	10:// homing sequence
		IF  Stop_PI = 0  THEN
			Out.Homed_PO :=0;
			//check this: reseting expected to match pulse count so that homeing will start if there is a mismatch
			//decide homing direction and homing method //make flag large enough to hit home switch and the limit switch
			IF IN.Limit_NC_NO_CI =0 THEN	//NC switch configuration
				IF bHigh_FI =1 AND bLow_FI =1 THEN	//using normally closed sensor (flag is not on either limit switch)
					IF IN.HomingSet_CI =2 THEN cw := 0; ELSIF IN.HomingSet_CI =3 THEN cw :=1; END_IF //go to high or low first if no limit switch tripped
				END_IF
			ELSE	//NO switch Configuration
				IF bHigh_FI =0 AND bLow_FI =0 THEN	//using normally closed sensor (flag is not on either limit switch)
					IF IN.HomingSet_CI =2 THEN cw := 0; ELSIF IN.HomingSet_CI =3 THEN cw :=1; END_IF //go to high or low first if no limit switch tripped
				END_IF
			END_IF
			//if inputA is hi then turn off (takes 2 cycles to output an increment at cp motor)
				(*if pulses expected = pulse count then do the next move *)
			IF AltSpeedCase = 60 THEN SendPulse(); END_IF
			IF IN.Limit_NC_NO_CI =0 THEN	//NC switch configuration
				IF bHome_FI =0 THEN //use nc switch for sensor [at home position]
					bHomeStart_PI :=0;
					Cancelmove();
					HomeCase := 20;
				END_IF
				ELSE				//NO switch configuration
				IF bHome_FI =1 THEN //use no switch for sensor [at home position]
				bHomeStart_PI :=0;
				Cancelmove();
				HomeCase := 20;
			END_IF	
			END_IF
			(*check this - add in an extra cycle before setting home that moves away from the 
				homed spot in same direction to confirm trigger positino comes on same side of sensor each time*)
		END_IF
	20:	//extra scan before homed
		HomeCase :=50;	//this scan is required to allow for a cancelled move reset after homing
	
	50://after homing reset motor and cancelled bit
		
			Out.Homed_PO := 1;
			//cancelled :=0;	//resets motor after initial homing
			pulsecount :=0;
			expectedPulse :=0;
			Out.DistancePos_PO :=0;
			Out.ExpDistancePos_PO :=0;
			testbool := TRUE;
			HomeCase := 0;	//back to the start
	90://reset to default or?
	
END_CASE
END_METHOD

METHOD PUBLIC InLimits : BOOL
VAR_INPUT
	Req	: REAL;	//reqested degree or position from abs move to be evaluated for limits
END_VAR
//only valid after homing
InLimits := TRUE;
IF IN.SWLimit_Hi_CI <=0 OR IN.SWLimit_Lo_CI >=0 THEN		//check this (may need to have a neg hi at some point)
	//message to say no limits are set
	InLimits :=FALSE;	
END_IF
IF Req <= IN.SWLimit_Hi_CI AND Req >= IN.SWLimit_Lo_CI THEN
	InLimits := TRUE;
	ELSE
		InLimits :=FALSE;
END_IF
END_METHOD

METHOD PUBLIC Jog : BOOL
VAR_INPUT
END_VAR

//add software limits check this
CASE JogCase OF 
	0:	//Main Jog Sequence [Also stops movement]
		IF JogSlow_VI THEN AltspeedReq :=1; ELSE AltSpeedReq :=0;   END_IF
			
		IF JogExecute_VI AND Out.Homed_PO =1  THEN	//if last move is done then allow for manual increment also required to be at home //check sensor check
			IF IN.Limit_NC_NO_CI = 0 THEN	//NC limit switch configuration
				IF bHigh_FI AND bLow_FI THEN //set direction via hmi unless on a limit switch then default to locateposition()
					IF CW_VI = 1 	THEN	CW := 1; 	ELSE CW:=0; 	END_IF
					IF bhigh_fI = 0	THEN 	CW:=0; 		END_IF
					IF bLow_FI = 0 	THEN 	CW:=1; 		END_IF
				END_IF
				ELSE	//NO limit switch configuration
					IF bHigh_FI =0 AND bLow_FI  = 0 THEN //set direction via hmi unless on a limit switch then default to locateposition()
					IF CW_VI = 1 	THEN	CW := 1; 	ELSE CW:=0; 	END_IF
					IF bhigh_fI = 1	THEN 	CW:=0; 		END_IF
					IF bLow_FI = 1 	THEN 	CW:=1; 		END_IF
				END_IF
			END_IF
			IF AltspeedReq THEN			// slowjog if altspeed is requested and wait for case 60
				IF AltspeedCase = 60 THEN
					SendPulse();
					
				END_IF
				ELSE
					SendPulse();		//send pulse for reg speed jog
			END_IF
			ELSE
				IF	JogExecute_VI  = FALSE THEN		
					CancelMove();
					JogCase :=10;
				END_IF
		END_IF
	10:	//
		IF JogExecute_VI =TRUE THEN JogCase :=0; END_IF
		
	
END_CASE
END_METHOD

METHOD PUBLIC LocatePosition : Bool //determines if sensorcheck is on and working.  Enables movement
VAR_INPUT
END_VAR

// Linear axis limit sensors
(*		bHigh_FI		AT %I*	: 	BOOL;
		bLow_FI			AT %I*	: 	BOOL;
		bHome_FI		AT %I*	: 	BOOL;*)
//NC limit sensor configuration
IF IN.Limit_NC_NO_CI = 0 THEN
	IF bHigh_FI =0 AND bInputBCom_FI =1 AND CW = 1 THEN	//use normally closed sensor and check inputb(-) [applies when trying to move past limit]
		cancelmove();
		CW := 0;	//require next move to be in Neg direction or CCW  //manual move will need to be used to get off limit switch check this
		//message saying that high limit as been exceeded or inputbcom is not connected
		Out.ErrorMsg_VO := 'High Limit reached, reset and move away from limit';
	END_IF
	IF bLow_FI =0 AND bInputBCom_FI = 0 AND CW =0 THEN	//use normally closed sensor and check inputb(-) [applies when trying to move past limit]
		cancelmove();
		CW :=1;	//require next move to be in Neg direction or CCW //manual move will need to be used to get off limit switch check this
		//message saying that Low limit as been exceeded or inputbcom is not connected
		Out.ErrorMsg_VO := 'Low Limit reached, reset and move away from limit';
	END_IF
ELSE
	//NO limit sensor configuration
	//additional option to use a N/O sensor if desired....not suggested
	IF bHigh_FI =1 AND bInputBCom_FI =1 AND CW = 1 THEN	//use normally closed sensor and check inputb(-) [applies when trying to move past limit]
		cancelmove();
		CW := 0;	//require next move to be in Neg direction or CCW  //manual move will need to be used to get off limit switch check this
		//message saying that high limit as been exceeded or inputbcom is not connected
		Out.ErrorMsg_VO := 'High Limit reached, reset and move away from limit';
	END_IF
	IF bLow_FI =1 AND bInputBCom_FI = 0 AND CW =0 THEN	//use normally closed sensor and check inputb(-) [applies when trying to move past limit]
		cancelmove();
		CW :=1;	//require next move to be in Neg direction or CCW //manual move will need to be used to get off limit switch check this
		//message saying that Low limit as been exceeded or inputbcom is not connected
		Out.ErrorMsg_VO := 'Low Limit reached, reset and move away from limit';
	END_IF
END_IF
Out.LastDistancePos_PO := Out.DistancePos_PO;
END_METHOD

METHOD PUBLIC MechDrive_CI : BOOL
VAR_INPUT
END_VAR
// 0: motor only(rot), 1: Motor and gear(rot), 2: Motor w/gear and screw(lin), 3: Motor w/screw only(lin), 4: Motor w/gear and pulley(lin),  5: Motor w/pulley(lin), 8: bypass mode
(*		DistPerMRev_CI		:	INT;	//distance traveled per rev		(Calculate your own pitch and lead w/gearbox combo must set MechDriveType_CI to 8 to bypass internal calc)
		DegPerMRev_CI		:	INT;	//distance traveled per rev		(Calculate your own pitch and lead w/gearbox combo must set MechDriveType_CI to 8 to bypass internal calc)
		DisPerFPulley_CI	:	INT;	//distance traveled per rev of final pulley (mm)
		GearRatio_CI		:	INT;	// GearRatio motor to moving part (XX:1) (gearbox and lead included in calc for vert axis) (use this for gearbox and pulleys as well)
		Lead_CI				:	INT;	// Lead of Screw if used (mm)			 (gearbox and lead included in calc for vert axis)	
*)

IF IN.MechDriveType_CI = 2 THEN	//2: Motor w/gear and screw(lin)
	DistPerMRev := IN.Lead_CI/IN.GearRatio_CI;	//driven mech ex 4mm/40 = .1mm per rev
	Out.MechTypeMsg_VO := 'Motor w/gear ratio and screw - no Degrees available [no rotary by default]';
	IF IN.GearRatio_CI <=0 OR IN.Lead_CI <=0 THEN
		isconfigured :=0;
		Out.MechTypeMsg_VO := 'GearRatio_CI or Lead_CI not configured please configure to continue';
	END_IF
END_IF

IF IN.MechDriveType_CI = 3 THEN	//3: Motor w/screw only(lin)
	DistPerMRev := IN.Lead_CI;		//driven mech ex 4mm = 4mm per rev
	Out.MechTypeMsg_VO := 'Motor w/screw - no Degrees available [no rotary by default]';
	IF IN.Lead_CI <=0 THEN
		isconfigured :=0;
		Out.MechTypeMsg_VO := 'Lead_CI not configured please configure to continue';
	END_IF
END_IF

IF IN.MechDriveType_CI = 4 THEN	//4: Motor w/gear and pulley(lin),
	DistPerMRev := IN.DisPerFPulley_CI/IN.GearRatio_CI;	//pulley circumference (20t at10 ~ 200mm per fin rev/gear ratio (40) = 5mm/motor rev
	Out.MechTypeMsg_VO := 'Motor w/gear ratio and pulley [no Degree used by default (linear pulley drive) if a rotary either use bypass or use type 1 and include pulley in gear ratio]';
	IF IN.GearRatio_CI <=0 OR IN.DisPerFPulley_CI <=0 THEN
		isconfigured :=0;
		Out.MechTypeMsg_VO := 'GearRatio_CI or DisPerFPulley_CI not configured please configure to continue';
	END_IF
END_IF

IF IN.MechDriveType_CI = 5 THEN	//5: Motor w/pulley(lin);
	DistPerMRev := IN.DisPerFPulley_CI;	//pulley circumference (20t at10 ~ 200mm per fin rev/gear ratio (40) = 5mm/motor rev
	Out.MechTypeMsg_VO := 'Motor w/pulley [no Degree used by default (linear pulley drive) if a rotary either use bypass or use type 1 and include pulley in gear ratio]';
	IF IN.DisPerFPulley_CI <=0 THEN
		isconfigured :=0;
		Out.MechTypeMsg_VO := 'DisPerFPulley_CI not configured please configure to continue';
	END_IF
END_IF

IF IN.MechDriveType_CI = 8 THEN	//8 mechdrivetype is bypassed and is set via DistPerMRev_CI or DegPerMRev_CI;
	DistPerMRev := IN.DistPerMRev_CI;
	Out.MechTypeMsg_VO := 'MechDriveType is bypassed - use DegPerMRev_CI or DistPerMRev_CI';
	IF IN.DistPerMRev_CI <=0  THEN
		isconfigured :=0;
		Out.MechTypeMsg_VO := 'DistPerMRev_CI not configured please configure to continue';
	END_IF
END_IF

IF IN.InputFilter_CI <=0 THEN
	isconfigured :=0;
	Out.ConfigMSG_VO := 'Input filter not configured, please check InputFilter_CI and clearpath motor settings';
END_IF

//linear axis
DisPerPulse := (DistPerMRev*IN.cntpulseSet_CI/32000);	//check this (Likely not a correct calc)
isConfigured :=1;	//sets configuration to true so that this block only runs once
END_METHOD

METHOD PUBLIC MoveAbsLin : BOOL
VAR_INPUT
		Req	: Real;	//input variable that will set FB DistancePosReq_PI
END_VAR
DistancePosReq_PI := Req;
DisToGo();
IF InLimits(DistancePosReq_PI) AND Out.Homed_PO =1 THEN //begin pulses
	IF PulsesEnabled =1 AND Stop_PI = 0 AND EnableOut_FO =1 AND CW = bInputBCom_FI THEN	//check for the motor being on before incrementing the distancepos from disreq	
		//if inputA is hi then turn off (takes 2 cycles to output an increment at cp motor)
		SendPulse();
	(*	IF InputAOut_FO =1 THEN 
			InputAOut_FO := 0;
			ELSE 
				InputAOut_FO :=1;		//else turn true and subtract increment counter
				MoveComplete :=0;		//Set movecomplete to zero until finished 
				Busy :=1;				//set busy until this pulse is complete (used to keep track of pos when using asg)
				IF CW=1 THEN DistancePos_PO := DistancePos_PO +1; 	ELSE DistancePos_PO := DistancePos_PO -1;	END_IF	//set distance movement based on directin moved		
				
			END_IF *)		
		ELSE
			error := 5;
		END_IF	
		//if input filter of clearpath is too high sometimes these pulses will not register (needed to maintain ability to chain moves)  Otherwise can use asg and movedone
	IF DistancePosReq_PI = Out.ExpDistancePos_PO AND MoveComplete =0 THEN 
		PulsesEnabled :=0; 
			//check this
	END_IF
ELSE
	//message not in limits	
END_IF
//add limits option here for stopping overtravel
END_METHOD

METHOD PUBLIC MoveDone : BOOL
VAR_INPUT
END_VAR
//ppr setting of hlfb is required
(*movecomplete is set either when pulsecount lines up exactly or if pulseque is empty and pulsecount is within tolerance*)
	IF PulseCount = expectedPulse  THEN	// (check this - add a tolerance here)
		MoveComplete :=1; 
		MoveDone := TRUE;
		busy :=0;			//set busy to zero (these are possibly interchangable until further code added) check this
		ELSE
			MoveDone :=FALSE;
		//is movedone() not completed check this
		//Add in MOVEDONE:=True; check this
	END_IF
	//movecomplete set for absolute move ppr tolerance
	IF PulseQueSet = 1 and PulseQue = 0 AND (pulseCount >= ExpectedPulse -2 OR PulseCount <= ExpectedPulse +2) THEN
		MoveComplete :=1;
		PulseQueSet :=0;
		MoveDone := TRUE;
		Busy :=0;
		//set expected to pulscount?
		//expectedPulse := PulseCount;
	END_IF
(* set DistPos_PO based off pulsecount/pulsecountset_ci  then check expectedDistPos_PO against current *)
//check busy and move complete in asg and if busytrig then check asgtrig then set move complete
END_METHOD

METHOD PUBLIC PPR : BOOL
VAR_INPUT
END_VAR
IF PulseCounter.Q THEN
	IF InputBOut_FO =1 THEN
		PulseCount := PulseCount +1;
		ELSE
			PulseCount := PulseCount -1;
		END_IF
		//extra pulse after homing is happening here? check this
END_IF

IF ATrig.Q AND Cancelled = 0 THEN
	IF InputBOut_FO = 1 THEN ExpectedPulse := ExpectedPulse + (1*IN.PPRset_CI); //does not account for cnt per rev yet
		ELSE ExpectedPulse := ExpectedPulse - (1*IN.PPRset_CI);
	END_IF
	//expectedpulse should be 32000cnts div by ppr = cnts per pulse
	//expectedPulse should be cntset_CI/320000 *(1*pprset_ci)   //30223cnts per pulse currently
END_IF
IF HomeTrig.Q THEN
	PulseCount  :=0;	//set position to zero after homing is complete
	ExpectedPulse := 0;
END_IF
IF Cancelled = 1 THEN
	expectedPulse := pulsecount;
END_IF
IF  movecomplete = 1 THEN //ppr mode
	 Out.DistancePos_PO := PulseCount/2; //change distancePOs_PO to float if needed
	 Out.ExpDistancePos_PO := PulseCount/2;
END_IF
IF  PowerOn_PI =0 THEN
	Out.DistancePos_PO := PulseCount/2; //change distancePOs_PO to float if needed	//resets DistancePos_PO if PowerOn_PI signal is interupted or turned off after if mid move
	 Out.ExpDistancePos_PO := PulseCount/2;
END_IF
Out.DistancePos_PO := PulseCount/2; //change distancePOs_PO to float if needed 
(* if expected pulses are in tolerance then pulsecount/ pprset should be used to set new dist position   
*)
END_METHOD

METHOD PUBLIC Reset : BOOL
VAR_INPUT
END_VAR
IF reset_VI =1 THEN
	EnableOut_FO :=0;	//Turn off to reset (power on will finish reset)
	Cancelled :=0;	//reset the cancelled move bit
	busy :=0;	// check this (is reseting busy needed?)
	Out.ErrorMsg_VO:= '';
	
End_if
//reset by turning power off and then on
END_METHOD

METHOD PUBLIC SendPulse : BOOL
VAR_INPUT
END_VAR
//got rid of 'and busy =0'
IF Stop_PI = 0  AND EnableOut_FO =1 AND CW = bInputBCom_FI THEN	//check for the motor being on before incrementing the distancepos from disreq	
	IF InputAOut_FO =1  THEN 
		InputAOut_FO := 0;
	ELSE 
		IF AltSpeedReq THEN
			IF AltspeedCase =60 THEN
				InputAOut_FO :=1;		//else turn true and subtract increment counter
				AltspeedCase :=0;	//reset altspeed
				IF CW =1 THEN Out.ExpDistancePos_PO := Out.ExpDistancePos_PO +1; ELSE Out.ExpDistancePos_PO := Out.ExpDistancePos_PO - 1; END_IF
			END_IF
		ELSE
			InputAOut_FO :=1;		//else turn true and subtract increment counter
			IF CW =1 THEN Out.ExpDistancePos_PO := Out.ExpDistancePos_PO +1; ELSE Out.ExpDistancePos_PO := Out.ExpDistancePos_PO - 1; END_IF
		END_IF
		MoveComplete :=0;		//set movedone to zero and await move complete
		busy		 :=1;		//set status to busy until move complete
	END_IF	
ELSE
	//InputAOut_FO := 0;		//no trigger if stopped or direction feedback failed or if motor enable is off
	//Message Saying Move is in progress
		
END_IF
END_METHOD

METHOD PUBLIC SuperJog : BOOL
VAR_INPUT
END_VAR
//using this mode will disable the two sensor safety check for manual manual mode
//homing is not required to use this and as such should be used with caution
//if not 2 sensors on and not in super mode then no movement allowed
	
	//message : at least one sensor is down please check sensors.  if movement is needed enter supermanual mode
	
//else  allow manual mode  even if not all sensors are working
	//message: you are in supermanual mode and will bypass anti collision devices.  please take caution
//add software limits check this

//add software limits check this
CASE SuperJogCase OF 
	0:	//Main Jog Sequence [Also stops movement]
		IF JogSlow_VI THEN AltspeedReq :=1; ELSE AltSpeedReq :=0;   END_IF
			
		IF SuperJogExecute_VI  THEN	//if last move is done then allow for manual increment also required to be at home //check sensor check
			(*IF IN.Limit_NC_NO_CI = 0 THEN	//NC limit switch configuration
				IF bHigh_FI AND bLow_FI THEN //set direction via hmi unless on a limit switch then default to locateposition()
					IF CW_VI = 1 	THEN	CW := 1; 	ELSE CW:=0; 	END_IF
					IF bhigh_fI = 0	THEN 	CW:=0; 		END_IF
					IF bLow_FI = 0 	THEN 	CW:=1; 		END_IF
				END_IF
				ELSE	//NO limit switch configuration
					IF bHigh_FI =0 AND bLow_FI  = 0 THEN //set direction via hmi unless on a limit switch then default to locateposition()
					IF CW_VI = 1 	THEN	CW := 1; 	ELSE CW:=0; 	END_IF
					IF bhigh_fI = 1	THEN 	CW:=0; 		END_IF
					IF bLow_FI = 1 	THEN 	CW:=1; 		END_IF
				END_IF
			END_IF*)
			IF CW_VI = 1 	THEN	CW := 1; 	ELSE CW:=0; 	END_IF
			IF AltspeedReq THEN			// slowjog if altspeed is requested and wait for case 60
				IF AltspeedCase = 60 THEN
					SendPulse();
					
				END_IF
				ELSE
					SendPulse();		//send pulse for reg speed jog
			END_IF
			ELSE
				IF	SuperJogExecute_VI  = FALSE THEN		
					CancelMove();
					SuperJogCase :=10;
				END_IF
		END_IF
	10:	//
		IF SuperJogExecute_VI =TRUE THEN SuperJogCase :=0; END_IF
		
	
END_CASE
END_METHOD

END_FUNCTION_BLOCK

// ---- Machine System/PRGs/Bogie/BogieCombo_PPR.TcPOU
FUNCTION_BLOCK BogieCombo_PPR
VAR_INPUT
	//Configuration Inputs
	VertSyncTolerance_CI 	: INT;
	Vert_A_CI				: LinPPR_CI;
	Vert_B_CI				: LinPPR_CI;
	Clamp_A_CI				: LinPPR_CI;
	Clamp_B_CI				: LinPPR_CI;
	
	
	//VI (visualization input/hmi input)
	Reset_VI				: BOOL;		//reset button		
	JogVertExecute_VI		: BOOL;		//Call manual vert move method if true
	JogClampExecute_VI		: BOOL;		//Call manual Clamp move method if true
	JogRotExecute_VI		: BOOL;		//Call manual Rot Move method if true
	SyncSuperJogExecute_VI	: BOOL;		//sync superjog manual move action bit
	SuperJogMode_VI			: BOOL;		//Superjog mode enable bit
	VertASuperJog_VI		: BOOL;
	VertBSuperJog_VI		: bool;		
	JogSlow_VI				: BOOL;		//slow manual move
	CW_VI					: BOOL;		//Set Direction for requested move (does not apply to absolute move) True = Clockwise
	SyncVertJogExecute_VI 	: BOOL;
	SyncClampJogExecute_VI 	: BOOL;

	//Program Inputs
	PowerOn_PI				: BOOL;
	VertDisReq_PI			: INT;
	ClampDisReq_PI			: INT;
	RotDegReq_PI			: INT;
	HomeWithPartStart_PI	: BOOL;		//set this true in program with oneshot to start homing, do not hold true in program as FB.Home() will continue to start at step 1
	SyncAbsDisReq_PI		: REAL;
	Stop_PI					: BOOL;		//stop command from program
	//Field Inputs
	PartPres_A_Hi			: BOOL;
	PartPres_A_Lo			: BOOL;
	PartPres_B_Hi			: BOOL;
	PartPres_B_Lo			: BOOL;
END_VAR
VAR_OUTPUT
	//Program OutPuts
	Homed_PO				: BOOL;	
	Msg						: STRING;	//debug message
END_VAR
VAR
	synctestbit				: bool;
	Vert_A					: ClearpathPositionLinPPR;
	Vert_B					: ClearpathPositionLinPPR;
	Clamp_A 				: ClearpathPositionLinPPR;
	Clamp_B					: ClearpathPositionLinPPR;
	Rot_A					: ClearpathPosition;
	Rot_B					: ClearpathPosition;
	
END_VAR
VAR PERSISTENT
	Vert_ATrack				: REAL;		//track the distance when not homed
	Vert_BTrack				: REAL;		//track the distance when not homed
	Clamp_ATrack			: REAL;		//track the distance when not homed
	Clamp_BTrack			: REAL;		//track the distance when not homed
	HomingReq				: BOOL;		//homing started, used to stop auto homing process if outside sync tolerance;  Superjog required to fix
END_VAR

//initialize the fb for bogie clearpaths bog[1-4 (vert, rot, clamp)
//Bog.Clamp();
//Bog.Rot();
Clamp_A	(IN:=Clamp_A_CI,Poweron_PI:=Poweron_pi, Stop_PI:=Stop_PI,Reset_VI:=Reset_VI, JogExecute_VI:=JogClampExecute_VI, JogSlow_VI:=JogSlow_VI, CW_VI:=CW_VI);
Clamp_B	(IN:=Clamp_B_CI,Poweron_PI:=Poweron_pi, Stop_PI:=Stop_PI,Reset_VI:=Reset_VI, JogExecute_VI:=JogClampExecute_VI, JogSlow_VI:=JogSlow_VI, CW_VI:=CW_VI);
Vert_A	(IN:=Vert_A_CI,Poweron_PI:=Poweron_pi, Stop_PI:=Stop_PI,Reset_VI:=Reset_VI, JogExecute_VI:=JogVertExecute_VI, JogSlow_VI:=JogSlow_VI, CW_VI:=CW_VI);
Vert_B	(IN:=Vert_B_CI,Poweron_PI:=Poweron_pi, Stop_PI:=Stop_PI,Reset_VI:=Reset_VI, JogExecute_VI:=JogVertExecute_VI, JogSlow_VI:=JogSlow_VI, CW_VI:=CW_VI);
//Rot_A();
//Rot_B();
//intialize the fb for bogie servo axis 1 and axis 2 in main pou	
//enable motors with enable hmi variable
If Vert_A.Out.Homed_PO=0 or Vert_B.Out.Homed_PO=0 then  Homed_PO:=0; End_if
//homing check

//SyncVertABSLin(VertDisReq_PI);
SuperMode(); 
HomeWithPart();
Syncvertjog();
(*8 From InSync() ..... Was being called every Insync() check but was not setting dis to lastdis*)
Vert_ATrack := Vert_ATrack + (Vert_A.Out.DistancePos_PO - Vert_A.Out.LastDistancePos_PO);
Vert_BTrack := Vert_BTrack + (Vert_B.Out.DistancePos_PO - Vert_B.Out.LastDistancePos_PO);
Clamp_ATrack := Clamp_ATrack + (Clamp_A.Out.DistancePos_PO - Clamp_A.Out.LastDistancePos_PO);
Clamp_BTrack := Clamp_BTrack + (Clamp_B.Out.DistancePos_PO - Clamp_B.Out.LastDistancePos_PO);
(* End From InSync()*)

//ready to receive move command

//move to request if above is met
IF InSync() = FALSE THEN
	IF SuperJogMode_VI =FALSE THEN	//if superjog mode is not enabled stop all moves if out of sync
		
	synctestbit :=1;
	Vert_A.CancelMove();
	Vert_B.CancelMove();
	Clamp_A.CancelMove();
	Clamp_B.CancelMove();
	msg := 'Not in Sync, Move Canceled, Reset and retry home';
	ELSE
		msg := ' SuperJog Mode in Progress, Caution';
	END_IF
END_IF

METHOD PUBLIC HomeSeparate : BOOL
VAR_INPUT
END_VAR
//if no tool is pressent then homing can be separate
t
END_METHOD

METHOD PUBLIC HomeWithPart : BOOL
VAR_INPUT
END_VAR
//if part present in one or both of the bogie verts then use this method

//set homepulsecountA from vert_a.pulsecount and use to avoid travel mismatch
//set homepulsecountB from vert_B.pulsecount and use to avoid travel mismatch

//Position Tracking
//after homingReq bit is true then
IF HomingReq THEN
	Vert_ATrack 	:= Vert_ATrack + (Vert_A.Out.DistancePos_PO - Vert_A.Out.LastDistancePos_PO);
	Vert_BTrack		:= Vert_BTrack + (Vert_B.Out.DistancePos_PO - Vert_B.Out.LastDistancePos_PO);
	Clamp_ATrack	:= Clamp_ATrack + (Clamp_A.Out.DistancePos_PO - Clamp_A.Out.LastDistancePos_PO);
	Clamp_BTrack	:= Clamp_BTrack + (Clamp_B.Out.DistancePos_PO -Clamp_B.Out.LastDistancePos_PO);
	ELSE 
		Vert_ATrack 	:=0;
		Vert_BTrack 	:=0;	
		Clamp_ATrack 	:=0;
		Clamp_BTrack 	:=0;
	END_IF

IF InSync() = FALSE AND SuperJogMode_VI = FALSE THEN
	//message not in sync	
	Vert_A.CancelMove();
	Vert_B.CancelMove();
	Clamp_A.CancelMove();
	Clamp_B.CancelMove();
	
END_IF

IF vert_A.Out.Homed_PO = 1 AND vert_B.out.Homed_PO =1 AND clamp_A.out.homed_po =1 AND clamp_b.Out.Homed_PO =1 THEN	//check for homed switch
	HomeWithPart:=TRUE;
	Homed_PO :=1;
	HomingReq :=0;
	ELSE
		HomeWithPart:=FALSE;
		Homed_PO :=0;
END_IF
IF HomeWithPartStart_PI = 1 THEN
	Vert_A.bHomeStart_PI := 1;
	Vert_B.bHomeStart_PI := 1;
	// dont home the clamps to the low sensor if part is present
	IF PartPres_A_Hi OR PartPres_A_Lo OR PartPres_B_Hi OR PartPres_B_lo THEN
		//message that part is present.  add to pressure and set home or leave same and set home
		
		ELSE
			Clamp_A.bHomeStart_PI := 1;
			Clamp_B.bHomeStart_PI := 1;
	END_IF
	//
	JogSlow_VI :=1;
	HomeWithPartStart_PI :=0;
	HomingReq :=1;
END_IF
	
//if homed on A and not B then keep pulsing B
	
	//if homed on B and not A then keep pulsing A
	
	//if not homed on A and B then pulse both again
	
	//wait pulse complete before sending another pulse
	//if homedswitch trig or limitswitch then cancelmove()
END_METHOD

METHOD PRIVATE InSync : BOOL
VAR_INPUT
END_VAR

IF Homed_PO THEN
	IF ABS(Vert_A.Out.DistancePos_PO - Vert_B.Out.DistancePos_PO) <= VertSyncTolerance_CI AND ABS(Clamp_A.Out.DistancePos_PO - Clamp_B.Out.DistancePos_PO) <= VertSyncTolerance_CI THEN
		InSync := TRUE;
	ELSE 
		InSync := FALSE;
	END_IF
ELSE
	IF ABS((Vert_ATrack) - (Vert_BTrack)) <= VertSyncTolerance_CI AND ABS((Clamp_ATrack) - (Clamp_BTrack)) <= VertSyncTolerance_CI THEN
			InSync := TRUE;
		ELSE
			InSync := FALSE;
	END_IF
END_IF
(*AND ABS((Clamp_ATrack) - (Clamp_BTrack)) <= VertSyncTolerance_CI*)
//add alarm and check this for when "InSync" is false and one motor has reached home switch and exceeds the sync tolerance
END_METHOD

METHOD Reset : BOOL
VAR_INPUT
END_VAR
END_METHOD

METHOD SuperMode : BOOL
VAR_INPUT
END_VAR
IF InSync()=TRUE AND SyncSuperJogExecute_VI AND SuperJogMode_VI THEN
	//jogs are canceled in 'ClearpathLinPPR' FB when SuperJogExecute is set to 0.
	Vert_A.SuperJogExecute_VI :=1;
	Vert_B.SuperJogExecute_VI :=1;
ELSE
	Vert_A.SuperJogExecute_VI :=0;
	Vert_B.SuperJogExecute_VI :=0;
END_IF

IF SuperJogMode_VI AND SyncSuperJogExecute_VI =0 THEN 	//sync move has to be off to move an individual
	Vert_A.SuperJogExecute_VI :=VertASuperJog_VI;
	Vert_B.SuperJogExecute_VI :=VertBSuperJog_VI;

END_IF
END_METHOD

METHOD SyncClampAbsLin : BOOL
VAR_INPUT
	req : REAL;
END_VAR
IF InSync()=TRUE  THEN
	Clamp_A.MoveAbsLin(Req);
	Clamp_B.MoveAbsLin(Req);
ELSE
	//re sync or cancel move
	Clamp_A.CancelMove();
	Clamp_B.CancelMove();
END_IF
END_METHOD

METHOD PUBLIC SyncVertAbsLin : BOOL
VAR_INPUT
	Req : REAL;
END_VAR
IF InSync()=TRUE  THEN
	Vert_A.MoveAbsLin(Req);
	Vert_B.MoveAbsLin(Req);
ELSE
	//re sync or cancel move
	Vert_A.CancelMove();
	Vert_B.CancelMove();
END_IF
END_METHOD

METHOD PRIVATE SyncVertJog : BOOL
VAR_INPUT
END_VAR
(*
IF InSync()=TRUE AND SyncJogExecute_VI THEN
	Vert_A.JogExecute_VI :=1;
	Vert_B.JogExecute_VI :=1;
ELSE
	Vert_A.JogExecute_VI :=0;
	Vert_B.JogExecute_VI :=0;
END_IF
*)
IF InSync()=TRUE AND SyncVertJogExecute_VI THEN
	JogVertExecute_VI :=1;
ELSE
	JogVertExecute_VI :=0;
END_IF
IF InSync()=TRUE AND SyncClampJogExecute_VI THEN
	JogClampExecute_VI :=1;
ELSE
	JogClampExecute_VI :=0;
END_IF
END_METHOD

END_FUNCTION_BLOCK

// ---- Machine System/PRGs/CAM_CNC/CNC/FB_SetAxisZero.TcPOU
FUNCTION_BLOCK FB_SetAxisZero
VAR_INPUT
	nHliAxisIdx: INT;
	bExecute: BOOL;
	bWriteOnStart: BOOL;
END_VAR
VAR_IN_OUT
	rOffset: LREAL;
END_VAR
VAR_OUTPUT
	bBusy: BOOL;
	bDone: BOOL;
	bError: BOOL;
END_VAR
VAR
	fbHLI3_SetAxisReferenceOffset : HLI3_SetAxisReferenceOffset;
	rtSetZero: R_TRIG;
	nCase: INT;
	rActPos: LREAL;
	bWriteOffset: BOOL;
	tmrWriteOffset: TON;
	rtWriteOffset: R_TRIG;
	rStartPos: LREAL;
	rOffsetValue: LREAL;
END_VAR

IF bDone AND NOT bExecute THEN
	bDone := FALSE;
END_IF

rtSetZero(CLK:= bExecute, Q=> );
IF rtSetZero.Q THEN
	bBusy := TRUE;
	bDone := FALSE;
	bError := FALSE;
	nCase := 10;
END_IF

tmrWriteOffset(IN:= bWriteOnStart, PT:= T#1S, Q=> , ET=> );
rtWriteOffset(CLK:= tmrWriteOffset.Q, Q=> );
IF rtWriteOffset.Q THEN
	IF rOffset <> 0 THEN
		bBusy := TRUE;
		bDone := FALSE;
		bError := FALSE;
		nCase := 110;
	ELSE
		nCase := 999;
	END_IF
END_IF

CASE nCase OF
	10:
		rOffsetValue := 0;
		bWriteOffset := TRUE;
		nCase := 20;
		
	20:
		IF NOT fbHLI3_SetAxisReferenceOffset.Error THEN
			IF fbHLI3_SetAxisReferenceOffset.Done THEN
				bWriteOffset := FALSE;
				nCase := 30;
			END_IF
		ELSE
			nCase := 999;
		END_IF
		
	30:
		rOffset := HLI3_GetActualAxisPos(nHliAxisIdx)*-0.0001;
		rOffsetValue := rOffset;
		nCase := 40;
		
	40:
		bWriteOffset := TRUE;
		nCase := 50;
		
	50:
		IF NOT fbHLI3_SetAxisReferenceOffset.Error THEN
			IF fbHLI3_SetAxisReferenceOffset.Done THEN
				bWriteOffset := FALSE;
				bBusy := FALSE;
				bDone := TRUE;
				nCase := 0;
			END_IF
		ELSE
			nCase := 999;
		END_IF
		
	999:
		bWriteOffset := FALSE;
		bBusy := FALSE;
		bError := TRUE;
		bDone := FALSE;
END_CASE

CASE nCase OF
	110:
		bWriteOffset := TRUE;
		rStartPos := HLI3_GetActualAxisPos(nHliAxisIdx)*0.0001;
		rOffsetValue := rOffset;
		nCase := 120;
		
	120:
		IF NOT fbHLI3_SetAxisReferenceOffset.Error THEN
			IF fbHLI3_SetAxisReferenceOffset.Done THEN
				bWriteOffset := FALSE;
				bBusy := FALSE;
				bError := FALSE;
				bDone := TRUE;
				nCase := 0;
			END_IF
		ELSE
			nCase := 999;
		END_IF
	
END_CASE

fbHLI3_SetAxisReferenceOffset(
	Execute:= bWriteOffset, 
	nHliAxisIdx:= nHliAxisIdx, 
	nOffset:= rOffsetValue, 
	Busy=> , 
	Done=> , 
	Error=> , 
	ErrorId=> );

END_FUNCTION_BLOCK

// ---- Machine System/PRGs/CAM_CNC/CNC/FB_StepperHomeToHardStop.TcPOU
FUNCTION_BLOCK FB_StepperHomeToHardStop
VAR_IN_OUT
	ax : axis_ref;
END_VAR
VAR_INPUT
	sEcatNetId : T_AmsNetId;  			// address of EtherCAT master the terminal is attached to
	nSlaveAddr: UINT;					// EtherCAT address of stepper terminal shown on EtherCAT tab of terminal
	bStartHome : BOOL;					// rising edge triggered
	iSetNormalMaxCurrent : INT;			// max current setting 
	iSetMaxHomeCurrent : INT;			// max current setting to use during home
	rHomePos: LREAL;					// positon of the axis when against the hard stop
	rHomeLagErrLimit: LREAL;			// lag error value to detect axis is against hard stop.  suggest as low a number as functionally possible (+5-10%).  If a value too low is used, you may need to go into the CoE paramaters and manually enter a larger number as the axis can fail due to overcurrnt fault on terminal
END_VAR
VAR_OUTPUT
	bBusy : BOOL;
	bErr : BOOL;
	bDone : BOOL;
END_VAR
VAR
	fbHome: MC_Home;
	fbReset: MC_Reset;
	fbJog: MC_Jog;
	fbSetPosition: MC_SetPosition;
	fbCoEWrite: FB_EcCoESdoWrite;
	fbCoERead: FB_EcCoESdoRead;
	fbWriteLimtMonitoring: MC_WriteBoolParameter;
	fbWriteLagMonitoring: MC_WriteBoolParameter;
	tmrDelay: TON;
	rtStartHome: R_TRIG;
	eHomeMode: MC_HomingMode;
	iMaxCurrentToSet : INT;
	iActMaxCurrent : INT;
	nCase: INT;
	nLastCase: INT;
	bResetAx: BOOL;
	bJogRev: BOOL;
	bJogFwd: BOOL;
	bWriteMaxCurrent: BOOL;
	bReadMaxCurrent: BOOL;
	bWriteLimitMonitoringValue: BOOL;
	bLimitMonitoringValue: BOOL;
	bWriteLagMonitoringValue: BOOL;
	bLagMonitoringValue: BOOL;
	bSetAxPosition: BOOL;
	bStartDelay: BOOL;
	bExecuteAxHome: BOOL;
	bJunkTrigger: BOOL;  // used for test when encoder was not present
END_VAR

(*
	This code is meant for a stepper terminal like EL7037 that has an encoder.  This will NOT work without a working configured encoder.  
	Use at your own risk....mechanical and electrical damage is possible!!
	
	This code will setp through homing a stepper motor to a hard stop.  Homing direction is negative (reverse).  Changing values in the NC axis for homing is ignored.
	
	Axis will move at the velocity set in axis parameter "Manual Velocity (Slow)" in NC configuration.
	
	Steps-
	-Write a max current value (value from FB input) to the stepper terminal that is just high enought to make the move
	-Disable lag error monitoring
	-Disable negative limit monitoring
	-Reset axis calibration flag to false
	-Jog in negative direction until following error exceeds a limit (value from FB input).  Jogs at axis slow speed jog setting in NC config
	-Stop
	-Reset
	-Write current position (value from FB input).  Recommend a value just less than zero, so axis can go to zero without risk of hitting hard stop
	-Enable lag error monitoring
	-Enable negative limit monitoring
	-Set axis calbration flag to true
	-Done
	
	If err occurs, look at nLastCase to determine what went wrong
*)

ax.ReadStatus();
	
tmrDelay(IN:= bStartDelay, PT:= T#500MS, Q=> , ET=> );

rtStartHome(CLK:= bStartHome, Q=> );

IF ax.Status.ControlLoopClosed AND rtStartHome.Q THEN
	bWriteMaxCurrent := FALSE;
	bReadMaxCurrent := FALSE;
	bWriteLimitMonitoringValue := FALSE;
	bWriteLagMonitoringValue := FALSE;
	bExecuteAxHome := FALSE;
	bStartDelay := FALSE;
	bJogFwd := FALSE;
	bJogRev := FALSE;
	bResetAx := FALSE;
	bSetAxPosition := FALSE;
	iActMaxCurrent := 0;
	bBusy := TRUE;
	bErr := FALSE;
	bDone := FALSE;
	nCase := 10;
END_IF

CASE nCase OF
	10:
		iMaxCurrentToSet := iSetMaxHomeCurrent;
		bWriteMaxCurrent := TRUE;
		nCase := 20;
		
	20: 
		IF NOT fbCoEWrite.bError THEN
			IF NOT fbCoEWrite.bBusy THEN
				bWriteMaxCurrent := FALSE;
				nCase := 30;
			END_IF
		ELSE 
			bErr := TRUE;
			nLastCase := nCase;
			nCase := 999;
		END_IF
		
	30:
		bReadMaxCurrent := TRUE;
		nCase := 40;
		
	40:
		IF NOT fbCoERead.bError THEN
			IF NOT fbCoERead.bBusy THEN
				bReadMaxCurrent := FALSE;
				nCase := 50;
			END_IF
		ELSE 
			bErr := TRUE;
			nLastCase := nCase;
			nCase := 999;
		END_IF
		
	50: 
		IF iSetMaxHomeCurrent = iActMaxCurrent THEN
			nCase := 60;
		ELSE 
			bErr := TRUE;
			nLastCase := nCase;
			nCase := 999;
		END_IF
		
	60:
		bLimitMonitoringValue := FALSE;
		bWriteLimitMonitoringValue := TRUE;
		bLagMonitoringValue := FALSE;
		bWriteLagMonitoringValue := TRUE;
		eHomeMode := MC_ResetCalibration;
		bExecuteAxHome := TRUE;
		nCase := 70;
		
	70:
		bWriteLimitMonitoringValue := FALSE;
		bWriteLagMonitoringValue := FALSE;
		bExecuteAxHome := FALSE;
		bStartDelay := TRUE;
		nCase := 80;
		
	80:
		IF tmrDelay.Q THEN
			bStartDelay := FALSE;
			bJogRev := TRUE;
			nCase := 90;
		END_IF
		
	90:
		IF (ABS(ax.NcToPlc.PosDiff) > rHomeLagErrLimit) OR bJunkTrigger THEN
			bJunkTrigger := FALSE;
			bJogRev := FALSE;
			bResetAx := TRUE;
			bStartDelay := TRUE;
			nCase := 100;
		END_IF
		
	100:
		IF tmrDelay.Q THEN
			bStartDelay := FALSE;
			bResetAx := FALSE;
			bSetAxPosition := TRUE;
			nCase := 110;
		END_IF
		
	110:
		bSetAxPosition := FALSE;
		nCase := 120;
		
	120:
		nCase := 130;
		
	130:
		IF (ax.NcToPlc.ActPos > (rHomePos - 0.005)) AND (ax.NcToPlc.ActPos < (rHomePos + 0.005)) THEN
			nCase := 140;
		END_IF
		
	140:
		iMaxCurrentToSet := iSetNormalMaxCurrent;
		bWriteMaxCurrent := TRUE;
		nCase := 150;
		
	150: 
		IF NOT fbCoEWrite.bError THEN
			IF NOT fbCoEWrite.bBusy THEN 
				bWriteMaxCurrent := FALSE;
				nCase := 160;
			END_IF
		ELSE 
			bErr := TRUE;
			nLastCase := nCase;
			nCase := 999;
		END_IF
		
	160:
		bReadMaxCurrent := TRUE;
		nCase := 170;
		
	170:
		IF NOT fbCoERead.bError THEN
			IF NOT fbCoERead.bBusy THEN
				bReadMaxCurrent := FALSE;
				nCase := 180;
			END_IF
		ELSE 
			bErr := TRUE;
			nLastCase := nCase;
			nCase := 999;
		END_IF
		
	180: 
		IF iMaxCurrentToSet = iActMaxCurrent THEN
			nCase := 190;
		ELSE 
			bErr := TRUE;
			nLastCase := nCase;
			nCase := 999;
		END_IF
		
	190:
		bLimitMonitoringValue := TRUE;
		bWriteLimitMonitoringValue := TRUE;
		bLagMonitoringValue := TRUE;
		bWriteLagMonitoringValue := TRUE;
		eHomeMode := MC_ForceCalibration;
		bExecuteAxHome := TRUE;
		nCase := 200;
		
	200:
		bWriteLimitMonitoringValue := FALSE;
		bWriteLagMonitoringValue := FALSE;
		bExecuteAxHome := FALSE;
		bDone := TRUE;
		IF NOT bStartHome THEN
			bBusy := FALSE;
			bDone := FALSE;
			nCase := 0;
		END_IF
		
	999:
		bWriteMaxCurrent := FALSE;
		bReadMaxCurrent := FALSE;
		bWriteLimitMonitoringValue := FALSE;
		bWriteLagMonitoringValue := FALSE;
		bExecuteAxHome := FALSE;
		bStartDelay := FALSE;
		bJogFwd := FALSE;
		bJogRev := FALSE;
		bResetAx := FALSE;
		bSetAxPosition := FALSE;
		bErr := TRUE;
		bDone := FALSE;
		nCase := 0;
		
END_CASE

fbCoEWrite(
	sNetId:= sEcatNetId, 
	nSlaveAddr:= nSlaveAddr, 
	nSubIndex:= 1, 
	nIndex:= 16#8010, 
	pSrcBuf:= ADR(iMaxCurrentToSet), 
	cbBufLen:= SIZEOF(iMaxCurrentToSet), 
	bExecute:= bWriteMaxCurrent, 
	tTimeout:= , 
	bBusy=> , 
	bError=> , 
	nErrId=> );
	
fbCoERead(
	sNetId:= sEcatNetId, 
	nSlaveAddr:= nSlaveAddr, 
	nSubIndex:= 1, 
	nIndex:= 16#8010, 
	pDstBuf:= ADR(iActMaxCurrent), 
	cbBufLen:= SIZEOF(iActMaxCurrent), 
	bExecute:= bReadMaxCurrent, 
	tTimeout:= , 
	bBusy=> , 
	bError=> , 
	nErrId=> );
	
fbWriteLimtMonitoring(
	Axis:= ax, 
	Execute:= bWriteLimitMonitoringValue, 
	ParameterNumber:= MC_AxisParameter.EnableLimitNeg, 
	Value:= bLimitMonitoringValue);
	
fbWriteLagMonitoring(
	Axis:= ax, 
	Execute:= bWriteLagMonitoringValue, 
	ParameterNumber:= MC_AxisParameter.EnablePosLagMonitoring, 
	Value:= bLagMonitoringValue);
	
fbSetPosition(
	Axis:= ax, 
	Execute:= bSetAxPosition, 
	Position:= rHomePos);
	
fbReset(
	Axis:= ax, 
	Execute:= bResetAx);

fbJog(
	Axis:= ax, 
	JogForward:= bJogFwd, 
	JogBackwards:= bJogRev);	
	
fbHome(
	Axis:= ax, 
	Execute:= bExecuteAxHome, 
	Position:= , 
	HomingMode:= eHomeMode);

END_FUNCTION_BLOCK

// ---- Machine System/PRGs/CAM_CNC/CNC/GetMotorTemps.TcPOU
PROGRAM GetMotorTemps
VAR
	tmrGetTemp: TON;
	fbGetMotorTemp: FB_EcCoESdoRead;
	arrMotorTemp : ARRAY[0..6] OF REAL;
	iSlaveAddr : UINT;
	iIndex : WORD;
	i : INT;
	X1MotorTemp : REAL;
	X2MotorTemp : REAL;
	YMotorTemp : REAL;
	ZMotorTemp : REAL;
	PMotorTemp : REAL;
END_VAR

	
tmrGetTemp(IN:= NOT tmrGetTemp.Q, PT:= T#10S, Q=> , ET=> );
IF tmrGetTemp.Q THEN
	i := i + 1;
	IF i > 5 THEN
		i := 0;
	END_IF
END_IF
		
IF i = 1 THEN
	iSlaveAddr := 1060; //X1
	iIndex := 16#32C1;
ELSIF i = 2 THEN
	iSlaveAddr := 1061; //X2
	iIndex := 16#32C1;
ELSIF i = 3 THEN
	iSlaveAddr := 1064; //Y
	iIndex := 16#32C1;
ELSIF i = 4 THEN
	iSlaveAddr := 1063; //Z
	iIndex := 16#36C1;
ELSIF i = 5 THEN
	iSlaveAddr := 1063; //Pallet
	iIndex := 16#32C1;
END_IF

fbGetMotorTemp(
	sNetId:= '169.254.21.118.3.1', 
	nSlaveAddr:= iSlaveAddr, 
	nSubIndex:= 6, 
	nIndex:= iIndex, 
	pDstBuf:= ADR(arrMotorTemp[i]), 
	cbBufLen:= SIZEOF(arrMotorTemp[i]), 
	bExecute:= tmrGetTemp.Q AND i<>0, 
	tTimeout:= , 
	bBusy=> , 
	bError=> , 
	nErrId=> );	

X1MotorTemp := arrMotorTemp[1];	
X2MotorTemp := arrMotorTemp[2];	
YMotorTemp := arrMotorTemp[3];	
ZMotorTemp := arrMotorTemp[4];	
PMotorTemp := arrMotorTemp[5];

END_PROGRAM

// ---- Machine System/PRGs/CAM_CNC/CNC/myBUTTONS.TcPOU
PROGRAM myBUTTONS
VAR
	rtHold: R_TRIG;
	bHoldCmd: bool;
	bRapidLed: BOOL;
END_VAR

PLCMachineMode[1].Start := bStartPB;
PLCMachineMode[1].Reset := bResetPB;

// Feedhold
bHoldLed := PLCMachineMode[0].ChannelSignals.FeedHold;
rtHold(CLK:= bHoldPB, Q=> );
IF rtHold.Q THEN
	bHoldCmd := NOT bHoldCmd;
END_IF
Global_HMI.PlcChannelSignals.FeedHold := bHoldCmd;

bRapidLed := stManualModeControlElements[0].stControlKeys[0].bKeyRapid;

PLCSpindleOverride := 50 + LREAL_TO_UINT(iSpindleOverridePot/32767.0*50.0); // limit overried to be 50% to 100?
IF PLCSpindleOverride > 99 THEN
	PLCSpindleOverride := 100;
ELSIF PLCSpindleOverride < 51 THEN
	PLCSpindleOverride := 50;
END_IF

PLCFeedOverride := 50 + LREAL_TO_UINT(iFeedrateOverridePot/32767.0*50.0); // limit overried to be 50% to 100?
IF PLCFeedOverride > 99 THEN
	PLCFeedOverride := 100;
ELSIF PLCFeedOverride < 51 THEN
	PLCFeedOverride := 50;
END_IF

END_PROGRAM

// ---- Machine System/PRGs/CAM_CNC/CNC/myHMIPLCRECIPE.TcPOU
PROGRAM myHMIPLCRECIPE
VAR
	cyc : st_manual;
	bCTest1 : BOOL;
END_VAR

IF cyc.cyl1 = 1 THEN
	bCTest1 := TRUE;
	ELSE bCTest1 := FALSE;
END_IF

END_PROGRAM

// ---- Machine System/PRGs/CAM_CNC/CNC/myMachine.TcPOU
PROGRAM myMachine
VAR
	fbEcat1: FB_EcDiagnostics;
	fbEcat3: FB_EcDiagnostics;
	Device1 AT %I*: AMSNETID;
	Device3 AT %I*: AMSNETID;
	fbGetCommandedSpindleRpm: FB_GetSpindleRpm;
	rX_PcsPos: DINT;
	howknows: UDINT;
	bTestG100 : BOOL;
	nCase : INT;
	bEnHBA : BOOL;
	
	bSendMessage : BOOL;
	bRaiseAlarm : BOOL;
	bConfirmAlarm : BOOL;
	bClearAlarm: BOOL;

	fbLogger : FB_TcEventLogger;
	fbMessage : FB_TcMessage;
	fbAlarm : FB_TcAlarm;
	bIsInitalized : BOOL;
	
	bSetJsonAttribute : BOOL;
	sJsonAttribute : STRING := '{"key":"value"}';
	
	hr : HRESULT;
	hrLastError : HRESULT;
	iCurrentMode : UDINT;
	iCurrentState : UDINT;
	bJunky : BOOL;
	rX_ActVel : LREAL;
	rY_ActVel : LREAL;
	rChActVel : LREAL;
	fbGetActiveGs: HLI3_GetChannelActiveG;
	bGetActiveGs : BOOL;
	stActiveGs : ARRAY[0..39] OF INT;
	tmrGetGs: TON;
	
	
	tmrGetTemp: TON;
	fbGetMotorTemp: FB_EcCoESdoRead;
	arrMotorTemp : ARRAY[0..6] OF REAL;
	iSlaveAddr : UINT;
	iIndex : WORD;
	i : INT;
END_VAR



// put at beginning of MAIN
fbEcat1(stAMSNETID:= Device1);
fbEcat3(stAMSNETID:= Device3);
	
IF NOT (fbEcat1.bInitComplete AND fbEcat3.bInitComplete) THEN 
	RETURN;
END_IF

mySafety();

(* just for reference to see axis data from PLC *)
	pX := gpAx[0]; 
	pY := gpAx[1]; 	
	pZ := gpAx[2];  
	pCh0 := gpCh[0];
	
	howknows := pCh0[0].mc_error.satz_r.kopf.error_id;
	
	iCurrentMode := HLI3_GetChannelMode(nChanIdx:= 0);
	iCurrentState := HLI3_GetChannelState(nChanIdx:= 0);
	
		
	rX_ActPos := HLI3_GetActualAxisPos(0); // or rX_ActPos := pX^.lr_state.current_position_acs_r*0.0001;
	rY_ActPos := HLI3_GetActualAxisPos(1);
	rZ_ActPos := HLI3_GetActualAxisPos(2);
	
	rX_PcsPos := pch0^.bahn_state.coord_r[0].act_position_r;
	rX_PcsPos := pch0^.bahn_state.coord_r[0].cmd_position_r;
	rX_ActVel :=  pch0^.bahn_state.coord_r[0].w0_velocity_r;
	rY_ActVel :=  pch0^.bahn_state.coord_r[1].w0_velocity_r;
	rChActVel := pch0^.bahn_state.active_feed_r;
	
	
// get S value of PLC controlled Spindle
fbGetCommandedSpindleRpm(
	nHliChannelIdx:= 0, 
	bChannelReset:= , 
	nRPM=> nCommandedRPM, 
	bError=> , 
	nErrorId=> );
	
myM_Codes();
//run a saved program in cnc from plc
IF bTestG100 AND PRG_CNCChannelHandler.CNCChannel[0].currentmode = 4 THEN
	bTestG100 := FALSE;
	nCase := 10;
END_IF

CASE nCase OF
	10:
		PLCMachineMode[0].MDI := TRUE;
		nCase := 20;
		
	20:
		IF PRG_CNCChannelHandler.CNCChannel[0].currentmode = 3 THEN
			PLCMachineMode[0].MDIString := 'L C:\CNC\G100test.nc';
			PLCMachineMode[0].Start := TRUE;
			nCase := 30;
		END_IF
	
	30:
		IF PRG_CNCChannelHandler.CNCChannel[0].currentstate = 4 THEN
			nCase := 40;
		END_IF
		
	40:
		IF PRG_CNCChannelHandler.CNCChannel[0].currentstate = 3 THEN
			PLCMachineMode[0].Manual := TRUE;
			nCase := 0;
		END_IF
END_CASE
PRG_ManualModeVirtualHBA(nChanIdx:= 0, bEnable:= bEnHBA, stManualModeParameter:= stManualModeParameter[0], stManualModeControlElements:= stManualModeControlElements[0]);
IF bJunky THEN
	bJunky := FALSE;
	HLI3_SetVEChannelLRealValue(
	nChanIdx:=0, 
	nVEIndex:=0, 
	nArrayIndex:=0, 
	bGlobal:=TRUE,
	val:=1);
END_IF
tmrGetGs(IN:= NOT tmrGetGs.Q, PT:= T#500MS, Q=> , ET=> );
fbGetActiveGs(
	bExec:= tmrGetGs.Q, 
	nChanIdx:= 0, 
	ActiveG=> stActiveGs, 
	bBusy=> , 
	bError=> , 
	nErrorID=> );
	
	
tmrGetTemp(IN:= NOT tmrGetTemp.Q, PT:= T#10S, Q=> , ET=> );
IF tmrGetTemp.Q THEN
	i := i + 1;
	IF i > 5 THEN
		i := 0;
	END_IF
END_IF
		
IF i = 1 THEN
	iSlaveAddr := 1060; //X1
	iIndex := 16#32C1;
ELSIF i = 2 THEN
	iSlaveAddr := 1061; //X2
	iIndex := 16#32C1;
ELSIF i = 3 THEN
	iSlaveAddr := 1064; //Y
	iIndex := 16#32C1;
ELSIF i = 4 THEN
	iSlaveAddr := 1063; //Z
	iIndex := 16#36C1;
ELSIF i = 5 THEN
	iSlaveAddr := 1063; //Pallet
	iIndex := 16#32C1;
END_IF

fbGetMotorTemp(
	sNetId:= '169.254.21.118.3.1', 
	nSlaveAddr:= iSlaveAddr, 
	nSubIndex:= 6, 
	nIndex:= iIndex, 
	pDstBuf:= ADR(arrMotorTemp[i]), 
	cbBufLen:= SIZEOF(arrMotorTemp[i]), 
	bExecute:= tmrGetTemp.Q AND i<>0, 
	tTimeout:= , 
	bBusy=> , 
	bError=> , 
	nErrId=> );

END_PROGRAM

// ---- Machine System/FBs/FB_EcDiagnostics.TcPOU
FUNCTION_BLOCK FB_EcDiagnostics
VAR_INPUT
	stAMSNETID : AMSNETID;
	bReset: BOOL;
END_VAR
VAR_OUTPUT
	bEcSlaveWarning: BOOL;
	sEcDiagErrMsg: STRING(255);
	bEcMasterError: BOOL;
	bEcSlaveError: BOOL;
	bFbErr: BOOL;
END_VAR
VAR
	stMasterStateHistoryMsg : ARRAY[0..99] OF STRING(255);
	stSlaveStateHistoryMsg : ARRAY[0..999] OF STRING(255);
	stEcConfSlaveInfo : ARRAY [0..EC_MAX_SLAVES] OF ST_EcSlaveConfigData;
	stEcSlaveCrcCounts : ARRAY[0..EC_MAX_SLAVES] OF DWORD;
	stEcSlaveStates : ARRAY[0..EC_MAX_SLAVES] OF ST_EcSlaveState;
	stLastSlaveState : ARRAY[0..EC_MAX_SLAVES] OF ST_EcSlaveState;
	stSlaveErr : ARRAY[0..EC_MAX_SLAVES] OF BOOL;
	sAMSNETID: STRING;
	bGetMasterState: BOOL;
	bGetConfiguredSlaveCount: BOOL;
	bGetActualSlaveCount: BOOL;
	bGetCrcCounts: BOOL;
	bGetEcFrameStats: BOOL;
	bGetSlaveStates: BOOL;
	fbEcGetMasterDevState: FB_EcGetMasterDevState;
	fbEcGetConfSlaves: FB_EcGetConfSlaves;
	fbEcGetSlaveCount: FB_EcGetSlaveCount;
	fbEcGetAllSlaveCrcErrors: FB_EcGetAllSlaveCrcErrors;
	fbEcMasterFrameStatistic: FB_EcMasterFrameStatistic;
	fbEcGetAllSlaveStates: FB_EcGetAllSlaveStates;
	fbEcMasterFrameStatisticClearCRC: FB_EcMasterFrameStatisticClearCRC;
	fbEcMasterFrameStatisticClearFrames: FB_EcMasterFrameStatisticClearFrames;
	fbEcMasterFrameStatisticClearTxRxErr: FB_EcMasterFrameStatisticClearTxRxErr;
	fbNT_GetTime: NT_GetTime;
	tmrGetTime : TON;
	tmrStarted: TON;
	rtStarted: R_TRIG;
	ftReset: F_TRIG;
	nLastCase: INT;
	nCase: INT;
	i: INT;
	iMasterStateHistoryMsgCount : INT;
	iSlaveStateHistoryMsgCount : INT;
	nLastMasterDevState: UINT;
	byNum : BYTE;
	stMasterDevState : ARRAY[0..3] OF BYTE;
	arrTempSlaveDevState : ARRAY[0..3] OF BYTE;
	sTempMasterStateMsg: STRING(255);
	sTempSlaveStateMsg: STRING(255);
	sTime : STRING;
	sMasterStateString: ARRAY[0..3] OF STRING;
	sSlaveStateString: ARRAY[0..3] OF STRING;
	stLastSlaveDevStateMsg : ARRAY[0..EC_MAX_SLAVES] OF STRING(255);
	bInitComplete : BOOL;
END_VAR

A_GetTime();

tmrStarted(IN:= TRUE, PT:= T#5S);
rtStarted(CLK:= tmrStarted.Q);
ftReset(CLK:= bReset);
IF rtStarted.Q OR ftReset.Q THEN
	nCase := 1;
END_IF

CASE nCase OF 
	1:
		nLastCase := 0;
		sEcDiagErrMsg := '';
		bGetMasterState := FALSE;
		iMasterStateHistoryMsgCount := 0;
		iSlaveStateHistoryMsgCount := 0;
		bGetConfiguredSlaveCount := FALSE;
		bGetActualSlaveCount := FALSE;
		bGetCrcCounts := FALSE;
		bEcSlaveWarning := FALSE;
		bGetEcFrameStats := FALSE;
		bGetSlaveStates := FALSE;
		bEcMasterError := FALSE;
		bEcSlaveError := FALSE;
		bFbErr := FALSE;
		MEMSET(ADR(stEcSlaveCrcCounts),0, SIZEOF(stEcSlaveCrcCounts));
		MEMSET(ADR(stSlaveErr),0, SIZEOF(stSlaveErr));
		MEMSET(ADR(stMasterStateHistoryMsg),0, SIZEOF(stMasterStateHistoryMsg));
		MEMSET(ADR(stSlaveStateHistoryMsg),0, SIZEOF(stSlaveStateHistoryMsg));
		MEMSET(ADR(stLastSlaveDevStateMsg),0, SIZEOF(stLastSlaveDevStateMsg));
		sAMSNETID := concat(BYTE_TO_STRING(stAMSNETID[0]),'.');
		sAMSNETID := concat(sAMSNETID,BYTE_TO_STRING(stAMSNETID[1]));
		sAMSNETID := concat(sAMSNETID,'.');
		sAMSNETID := concat(sAMSNETID,BYTE_TO_STRING(stAMSNETID[2]));
		sAMSNETID := concat(sAMSNETID,'.');
		sAMSNETID := concat(sAMSNETID,BYTE_TO_STRING(stAMSNETID[3]));
		sAMSNETID := concat(sAMSNETID,'.');
		sAMSNETID := concat(sAMSNETID,BYTE_TO_STRING(stAMSNETID[4]));
		sAMSNETID := concat(sAMSNETID,'.');
		sAMSNETID := concat(sAMSNETID,BYTE_TO_STRING(stAMSNETID[5]));
		bInitComplete := FALSE;
		nCase := 10;
		
		
	10:
		bGetConfiguredSlaveCount := TRUE;
		nCase := 20;
		
	20:
		bGetConfiguredSlaveCount := FALSE;
		IF NOT fbEcGetConfSlaves.bError THEN
			IF NOT fbEcGetConfSlaves.bBusy THEN
				nCase := 30;
			END_IF
		ELSE
			bFbErr := TRUE;
			nLastCase := nCase;
			nCase := 30;
			sEcDiagErrMsg := 'Getting Master Configured Slave Count Failed';
		END_IF		
		
	30:
		bGetMasterState := TRUE;
		nCase := 40;
		
	40:
		bGetMasterState := FALSE;
		IF NOT fbEcGetMasterDevState.bError THEN
			IF NOT fbEcGetMasterDevState.bBusy THEN
				nCase := 50;
			END_IF
		ELSE
			bFbErr := TRUE;
			nLastCase := nCase;
			nCase := 50;
			sEcDiagErrMsg := 'Getting Master State failed';
		END_IF
		
	50:
		A_MasterStateMsg();
		nCase := 60;

	60:
		bGetActualSlaveCount := TRUE;
		nCase := 70;
		
	70:
		bGetActualSlaveCount := FALSE;
		IF NOT fbEcGetSlaveCount.bError THEN
			IF NOT fbEcGetSlaveCount.bBusy THEN
				nCase := 80;
			END_IF
		ELSE
			bFbErr := TRUE;
			nLastCase := nCase;	
			nCase := 80;
			sEcDiagErrMsg := 'Getting Master Actual Slave Count Failed';
		END_IF
		
	80:
		IF fbEcGetConfSlaves.nSlaves <> fbEcGetSlaveCount.nSlaves THEN
			bEcSlaveError := TRUE;
			nLastCase := nCase;
			sEcDiagErrMsg := 'Actual Slave Count <> Configured Slave Count';
		END_IF
		nCase := 90;
		
	90:
		bGetCrcCounts := TRUE;
		nCase := 100;
		
	100:
		bGetCrcCounts := FALSE;
		IF NOT fbEcGetAllSlaveCrcErrors.bError THEN
			IF NOT fbEcGetAllSlaveCrcErrors.bBusy THEN
				nCase := 110;
			END_IF
		ELSE
			bFbErr := TRUE;
			nLastCase := nCase;
			nCase := 110;
			sEcDiagErrMsg := 'Getting Slave CRC counts failed';
		END_IF
	
	110:
		FOR i := 0 TO (fbEcGetConfSlaves.nSlaves - 1) BY 1 DO
			IF stEcSlaveCrcCounts[i] > 0 THEN
				bEcSlaveWarning := TRUE;
				sEcDiagErrMsg := 'CRC counts on slaves';
			END_IF
		END_FOR
		nCase := 120;
		
	120:
		bGetEcFrameStats := TRUE;
		nCase := 130;
		
	130:
		bGetEcFrameStats := FALSE;
		IF NOT fbEcMasterFrameStatistic.bError THEN
			IF NOT fbEcMasterFrameStatistic.bBusy THEN
				nCase := 140;
			END_IF
		ELSE
			bFbErr := TRUE;
			nLastCase := nCase;
			nCase := 140;
		END_IF
		
	140:
		IF fbEcMasterFrameStatistic.nLostFrames > 2 OR fbEcMasterFrameStatistic.nLostQueuedFrames > 2 THEN
				bEcSlaveWarning := TRUE;
				sEcDiagErrMsg := 'Lost EtherCAT frames';
		END_IF
		nCase := 150;
		
	150:
		bGetSlaveStates := TRUE;
		nCase := 160;
		
	160:
		bGetSlaveStates := FALSE;
		IF NOT fbEcGetAllSlaveStates.bError THEN
			IF NOT fbEcGetAllSlaveStates.bBusy THEN
				nCase := 170;
			END_IF
		ELSE
			bFbErr := TRUE;
			nLastCase := nCase;
			nCase := 170;
			sEcDiagErrMsg := 'Getting Slave States failed';
		END_IF
		
	170:
		bInitComplete := TRUE;
		A_SlaveStateMsg();
		nCase := 30;
		
END_CASE

fbEcGetMasterDevState(
	sNetId:= sAMSNETID, 
	bExecute:= bGetMasterState);
	
fbEcGetConfSlaves(
	sNetId:= sAMSNETID, 
	pArrEcConfSlaveInfo:= ADR(stEcConfSlaveInfo), 
	cbBufLen:= SIZEOF(stEcConfSlaveInfo), 
	bExecute:= bGetConfiguredSlaveCount);
	
fbEcGetSlaveCount(
	sNetId:= sAMSNETID, 
	bExecute:= bGetActualSlaveCount);
	
fbEcGetAllSlaveCrcErrors(
	sNetId:= sAMSNETID, 
	pCrcErrorBuf:= ADR(stEcSlaveCrcCounts), 
	cbBufLen:= fbEcGetConfSlaves.nSlaves * 4, 
	bExecute:= bGetCrcCounts);
	
fbEcMasterFrameStatistic(
	sNetId:= sAMSNETID, 
	bExecute:= bGetEcFrameStats);
	
fbEcGetAllSlaveStates(
	sNetId:= sAMSNETID, 
	pStateBuf:= ADR(stEcSlaveStates), 
	cbBufLen:= SIZEOF(stEcSlaveStates), 
	bExecute:= bGetSlaveStates);
	
fbEcMasterFrameStatisticClearCRC(
	sNetId:= sAMSNETID, 
	bExecute:= bReset);
	
fbEcMasterFrameStatisticClearFrames(
	sNetId:= sAMSNETID, 
	bExecute:= bReset);
	
fbEcMasterFrameStatisticClearTxRxErr(
	sNetId:= , 
	nEcMasterDevID:= stAMSNETID[4] - 1, 
	bExecute:= bReset);
	
IF fbEcMasterFrameStatisticClearCRC.bError OR fbEcMasterFrameStatisticClearFrames.bError OR fbEcMasterFrameStatisticClearTxRxErr.bError THEN
	bFbErr := TRUE;
	sEcDiagErrMsg := 'Clearing CRC/TxRx Stats failed';
END_IF

ACTION A_GetTime:
tmrGetTime(IN := NOT tmrGetTime.Q, PT := T#20MS);
fbNT_GetTime(
	START:= tmrGetTime.Q,
	TMOUT:= T#1S);
	sTime:= WORD_TO_STRING(fbNT_GetTime.TIMESTR.wMonth);
	sTime:= CONCAT(sTime,'-' );
	sTime:= CONCAT(sTime, (WORD_TO_STRING(fbNT_GetTime.TIMESTR.wDay)));
	sTime:= CONCAT(sTime,'-' );
	sTime:= CONCAT(sTime, (WORD_TO_STRING(fbNT_GetTime.TIMESTR.wYear)));
	sTime:= CONCAT(sTime,'@' );
	sTime:= CONCAT(sTime, (WORD_TO_STRING(fbNT_GetTime.TIMESTR.wHour)));
	sTime:= CONCAT(sTime,':' );
	sTime:= CONCAT(sTime, (WORD_TO_STRING(fbNT_GetTime.TIMESTR.wMinute)));
	sTime:= CONCAT(sTime,':' );
	sTime:= CONCAT(sTime, (WORD_TO_STRING(fbNT_GetTime.TIMESTR.wSecond)));
	sTime:= CONCAT(sTime,':' );
	sTime:= CONCAT(sTime, (WORD_TO_STRING(fbNT_GetTime.TIMESTR.wMilliseconds)));
	sTime:= CONCAT(sTime,'ms ' );
END_ACTION

ACTION A_MasterStateMsg:

stMasterDevState[0] := WORD_TO_BYTE(ROL(fbEcGetMasterDevState.nDevState, 4))/16;
stMasterDevState[1] := WORD_TO_BYTE(fbEcGetMasterDevState.nDevState)/16;
stMasterDevState[2] := WORD_TO_BYTE(ROL(fbEcGetMasterDevState.nDevState, 12))/16;
stMasterDevState[3] := WORD_TO_BYTE(ROL(fbEcGetMasterDevState.nDevState, 8))/16;

(*0x1000 = DC not in sync *)
IF        stMasterDevState[3] = 0 THEN
		sMasterStateString[3] := '';
ELSIF     stMasterDevState[3] = 1 THEN
		sMasterStateString[3] := 'DC not in sync, ';
ELSE
		sMasterStateString[3] := 'Unknown error, ';
END_IF

(* 0x0100 = At least one device in 'INIT' state, 0x0200 = At least one device in 'PRE-OP' state, 0x0400 = At least one device in 'SAFE-OP' state, 0x0800 = At least one device indicates an error state *)
IF        stMasterDevState[2] = 0 THEN
		sMasterStateString[2] := '';
ELSIF     stMasterDevState[2] = 1 THEN
		sMasterStateString[2] := 'At least one device in INIT state, ';
ELSIF     stMasterDevState[2] = 2 THEN
		sMasterStateString[2] := 'At least one device in PREOP state, ';
ELSIF     stMasterDevState[2] = 4 THEN
		sMasterStateString[2] := 'At least one device in SAFE-OP state, ';
ELSIF     stMasterDevState[2] = 8 THEN
		sMasterStateString[2] := 'At least one device indicates an error state, ';
ELSE
		sMasterStateString[2] := 'Unknown error, ';
END_IF

(* 0x0010 = Out of send resources (I/O reset required), 0x0020 = Watchdog triggered, 0x0040 = Ethernet driver (miniport) not found, 0x0080 = I/O reset active *)
IF        stMasterDevState[1] = 0 THEN
		sMasterStateString[1] := '';
ELSIF     stMasterDevState[1] = 1 THEN
		sMasterStateString[1] := 'Out of send resources (I/O reset required), ';
ELSIF     stMasterDevState[1] = 2 THEN
		sMasterStateString[1] := 'Watchdog triggered, ';
ELSIF     stMasterDevState[1] = 4 THEN
		sMasterStateString[1] := 'Ethernet driver (miniport) not found, ';
ELSIF     stMasterDevState[1] = 8 THEN
		sMasterStateString[1] := 'I/O reset active, ';
ELSE
		sMasterStateString[1] := 'Unknown error, ';
END_IF

(* 0x0001 = Link error, 0x0002 = I/O locked after link error (I/O reset required), 0x0004 = Link error (redundancy adapter), 0x0008 = Missing one frame (redundancy mode) *)
IF        stMasterDevState[0] = 0 THEN
		sMasterStateString[0] := 'No Error.';
ELSIF     stMasterDevState[0] = 1 THEN
		sMasterStateString[0] := 'Link error.';
ELSIF     stMasterDevState[0] = 2 THEN
		sMasterStateString[0] := 'I/O locked after link error (I/O reset required).';
ELSIF     stMasterDevState[0] = 4 THEN
		sMasterStateString[0] := 'Link error (redundancy adapter).';
ELSIF     stMasterDevState[0] = 8 THEN
		sMasterStateString[0] := 'Missing one frame (redundancy mode).';
ELSE
		sMasterStateString[0] := 'Unknown error, ';
END_IF

IF fbEcGetMasterDevState.nDevState <> nLastMasterDevState THEN
	nLastMasterDevState := fbEcGetMasterDevState.nDevState;
	IF stMasterDevState[0] <> 0 THEN
		bEcMasterError := TRUE;
	END_IF
	IF stMasterStateHistoryMsg[iMasterStateHistoryMsgCount] = '' THEN
		sTempMasterStateMsg := sTime;
		sTempMasterStateMsg := concat(sTempMasterStateMsg, ' Master is ');
		sTempMasterStateMsg := concat(sTempMasterStateMsg, sMasterStateString[3]);
		sTempMasterStateMsg := concat(sTempMasterStateMsg, sMasterStateString[2]);
		sTempMasterStateMsg := concat(sTempMasterStateMsg, sMasterStateString[1]);
		sTempMasterStateMsg := concat(sTempMasterStateMsg, sMasterStateString[0]);
		stMasterStateHistoryMsg[iMasterStateHistoryMsgCount] := sTempMasterStateMsg;
		iMasterStateHistoryMsgCount := iMasterStateHistoryMsgCount + 1;
		IF iMasterStateHistoryMsgCount > 99 THEN
			iMasterStateHistoryMsgCount := 0;
		END_IF
	END_IF
END_IF
END_ACTION

ACTION A_SlaveStateMsg:

FOR i := 0 TO (fbEcGetConfSlaves.nSlaves - 1) BY 1 DO
	arrTempSlaveDevState[0] := ROL(stEcSlaveStates[i].deviceState,4)/16; 
	arrTempSlaveDevState[1] := stEcSlaveStates[i].deviceState/16;
	arrTempSlaveDevState[2] := ROL(stEcSlaveStates[i].linkState,4)/16;
	arrTempSlaveDevState[3] := stEcSlaveStates[i].linkState/16;
	
	(* 0x100_ = Communication port A, 0x200_ = Communication port B, 0x400_ = Communication port C, 0x800_ = Communication port D *)
	IF    arrTempSlaveDevState[3] = 0 THEN
			sSlaveStateString[3] := '';
	ELSIF arrTempSlaveDevState[3] = 1 THEN
			sSlaveStateString[3] := 'Comm Port A error, ';
	ELSIF arrTempSlaveDevState[3] = 2 THEN
			sSlaveStateString[3] := 'Comm Port B error, ';
	ELSIF arrTempSlaveDevState[3] = 4 THEN
			sSlaveStateString[3] := 'Comm Port C error, ';
	ELSIF arrTempSlaveDevState[3] = 8 THEN
			sSlaveStateString[3] := 'Comm Port D error, ';
	ELSE
			sSlaveStateString[3] := 'Unknown error, ';
	END_IF
	
	(* 0x010_ = Slave not present, 0x020_ = Slave signals link error, 0x040_ = Slave signals missing link, 0x080_ = Slave signals unexpected link *)	
	IF    arrTempSlaveDevState[2] = 0 THEN
			sSlaveStateString[2] := '';
	ELSIF arrTempSlaveDevState[2] = 1 THEN
			sSlaveStateString[2] := 'Slave not present, ';
	ELSIF arrTempSlaveDevState[2] = 2 THEN
			sSlaveStateString[2] := 'Slave signals link error, ';
	ELSIF arrTempSlaveDevState[2] = 4 THEN
			sSlaveStateString[2] := 'Slave signals missing link, ';
	ELSIF arrTempSlaveDevState[2] = 8 THEN
			sSlaveStateString[2] := 'Slave signals unexpected link, ';
	ELSE
			sSlaveStateString[2] := 'Unknown error, ';
	END_IF	
		
	(* 0x001_ = Slave signals error, 0x002_ = Invalid vendorId, productCode... read, 0x004_ = Initialization error occurred, 0x008_ = Slave disabled *)
	IF    arrTempSlaveDevState[1] = 0 THEN
			sSlaveStateString[1] := '';
	ELSIF arrTempSlaveDevState[1] = 1 THEN
			sSlaveStateString[1] := 'Slave signals error, ';
	ELSIF arrTempSlaveDevState[1] = 2 THEN
			sSlaveStateString[1] := 'Invalid vendorId - productCode... read, ';
	ELSIF arrTempSlaveDevState[1] = 4 THEN
			sSlaveStateString[1] := 'Initialization error occurred, ';
	ELSIF arrTempSlaveDevState[1] = 8 THEN
			sSlaveStateString[1] := 'Slave disabled, ';
	ELSE
			sSlaveStateString[1] := 'Unknown error, ';
	END_IF	
	
	(* 0x___1 = Slave in 'INIT' state, 0x___2 = Slave in 'PREOP' state, 0x___3 = Slave in 'BOOT' state, 0x___4 = Slave in 'SAFEOP' state, 0x___8 = Slave in 'OP' state *)
	IF    arrTempSlaveDevState[0] = 0 THEN
			sSlaveStateString[0] := '';
	ELSIF arrTempSlaveDevState[0] = 1 THEN
			sSlaveStateString[0] := 'INIT state.';
	ELSIF arrTempSlaveDevState[0] = 2 THEN
			sSlaveStateString[0] := 'PREOP state.';
	ELSIF arrTempSlaveDevState[0] = 3 THEN
			sSlaveStateString[0] := 'BOOT state.';
	ELSIF arrTempSlaveDevState[0] = 4 THEN
			sSlaveStateString[0] := 'SAFEOP state.';
	ELSIF arrTempSlaveDevState[0] = 8 THEN
			sSlaveStateString[0] := 'OP state.';
	ELSE
			sSlaveStateString[0] := 'Unknown State.';
	END_IF	
	
	sTempSlaveStateMsg := sTime;
	sTempSlaveStateMsg := concat(sTempSlaveStateMsg, stEcConfSlaveInfo[i].sName);
	sTempSlaveStateMsg := concat(sTempSlaveStateMsg, ' Slave is ');
	sTempSlaveStateMsg := concat(sTempSlaveStateMsg, sSlaveStateString[3]);
	sTempSlaveStateMsg := concat(sTempSlaveStateMsg, sSlaveStateString[2]);
	sTempSlaveStateMsg := concat(sTempSlaveStateMsg, sSlaveStateString[1]);
	sTempSlaveStateMsg := concat(sTempSlaveStateMsg, sSlaveStateString[0]);
	IF (stLastSlaveState[i].deviceState <> stEcSlaveStates[i].deviceState) OR (stLastSlaveState[i].linkState <> stEcSlaveStates[i].linkState) THEN
		stLastSlaveState[i].linkState := stEcSlaveStates[i].linkState;
		stLastSlaveState[i].deviceState := stEcSlaveStates[i].deviceState;
		stLastSlaveDevStateMsg[i] := sTempSlaveStateMsg;
		stSlaveStateHistoryMsg[iSlaveStateHistoryMsgCount] := sTempSlaveStateMsg;
		iSlaveStateHistoryMsgCount := iSlaveStateHistoryMsgCount + 1;
		IF iSlaveStateHistoryMsgCount > 999 THEN
			iSlaveStateHistoryMsgCount := 0;
		END_IF
	END_IF
	IF (stEcSlaveStates[i].deviceState <> 8) OR (stEcSlaveStates[i].linkState <> 0) THEN
		bEcSlaveError := TRUE;
		stSlaveErr[i] := TRUE;
		IF NOT bEcMasterError THEN
			sEcDiagErrMsg := sTempSlaveStateMsg;
		END_IF
	ELSE
		stSlaveErr[i] := FALSE;
	END_IF
END_FOR
END_ACTION

END_FUNCTION_BLOCK

// ---- Machine System/FBs/FB_GetSpindleRpm.TcPOU
FUNCTION_BLOCK FB_GetSpindleRpm
VAR_INPUT
	nHliChannelIdx: INT;	
	bChannelReset: BOOL;
END_VAR
VAR_OUTPUT
	nRPM : DINT;
	bError: BOOL;
	nErrorId: UDINT;
END_VAR
VAR		
	nHliAxisIdx: INT;
	bIsChannelSpecific: BOOL;	
	nOpenTechnoCount: UINT;	
	bAcknowledge: BOOL;
	nHliAxIfcIdx: UDINT;
	nTechFctMaxIdx: UINT;
	nLoop: UINT;
	pActTechnoUnit: POINTER TO TECHNO_UNIT_AX;
	pSProcess: POINTER TO HLI_S_PROZESS;
	pMProcess: POINTER TO HLI_M_H_PROZESS;
	fbRtrigChannelReset: R_TRIG;
	nLastRPM: DINT;
END_VAR


(****************************************************************************************)
(*							  Check for valid logical axis no.							*)
(****************************************************************************************)
IF NOT HLI3_CheckAxisValid(nHliAxisIdx := nHliAxisIdx) THEN
	bError									:= TRUE;
	nErrorId								:= 10000;
	RETURN;
END_IF

IF NOT HLI3_CheckChannelValid(nChannel := nHliChannelIdx) THEN
	bError									:= TRUE;
	nErrorId								:= 20000;
	RETURN;	
END_IF

(****************************************************************************************)
(*											Reset										*)
(****************************************************************************************)
fbRtrigChannelReset
	(CLK := bChannelReset);

IF fbRtrigChannelReset.Q THEN
	bAcknowledge	:= FALSE;
END_IF

(****************************************************************************************)
(*									Receive requests from cnc							*)
(****************************************************************************************)
(* Look out for open technology function either on the channel or the axis specific		*)
(* section of the HLI, depending on parameter ''.										*)
IF bIsChannelSpecific THEN
	nOpenTechnoCount	:= gpCh[nHliChannelIdx]^.used_units_std_sync_r;
	nTechFctMaxidx 		:= gpCh[nHliChannelIdx]^.used_units_std_sync_r - 1;
ELSE
	nOpenTechnoCount	:= gpAx[nHliAxisIdx]^.used_units_std_sync_r;
	nTechFctMaxidx 		:= gpAx[nHliAxisIdx]^.used_units_std_sync_r - 1;
END_IF

IF nOpenTechnoCount > 0 THEN
	FOR nLoop := 0 TO nTechFctMaxIdx DO
		(* Depending on the source determined by parameter 'bIsChannelSpecific', the		*)
		(* channel or axis specific section of the HLI will be examined.					*)
		IF bIsChannelSpecific THEN
			pActTechnoUnit	:= ADR(gpCh[nHliChannelIdx]^.techno_unit_std_sync[nLoop]);
		ELSE
			(* Get current axis specifc technology data *)
			pActTechnoUnit	:= ADR(gpAx[nHliAxisIdx]^.techno_unit_std_sync[nLoop]);
		END_IF
		

		(* Check request *)
		IF pActTechnoUnit^.please_rw AND
		   NOT pActTechnoUnit^.done_w
		THEN
			CASE UINT_TO_UDINT(pActTechnoUnit^.fkt_ctrl_r) OF
		     (* -------------------------------------------------------------------------- *)
			 (* Handle M function *)
			 HLI_INTF_M_FKT:
				pMProcess					:= ADR(pActTechnoUnit^.attribut_r.data[0]);
				
				
			 (* -------------------------------------------------------------------------- *)
			 (* Handle S function *)
			 HLI_INTF_SPINDEL:
				pSProcess					:= ADR(pActTechnoUnit^.attribut_r.data[0]);
				nRPM := pSProcess^.rev/6000;
				(* If we are working with spindle functions provided by the channel 		*)
				(* specific section of the HLI the logical axis number transmitted from the *)
				(* CNC must fit the one given in parameter 'nLogAxisNo'!					*)												
				IF bIsChannelSpecific AND (pSProcess^.log_achs_nr <> INT_TO_UINT(HLI3_GetLogAxisId(nHliAxisIdx:=nHliAxisIdx))) THEN
					RETURN;
				END_IF
	
			END_CASE
	
			(* Handle acknowledgement *)
			IF bAcknowledge THEN
				bAcknowledge				:= FALSE;
				pActTechnoUnit^.please_rw 	:= FALSE;
		   		pActTechnoUnit^.done_w		:= TRUE;
			END_IF
		END_IF
	END_FOR

END_IF
bIsChannelSpecific := TRUE;
IF nLastRPM <> nRPM THEN
	nLastRPM := nRPM;
	bIsChannelSpecific := FALSE;
END_IF

METHOD PRIVATE M_ManageAcknowledgement
VAR_INPUT
	pInternal			: POINTER TO BOOL;
	pPublic				: POINTER TO BOOL;
	pAcknowledgement	: POINTER TO BOOL;
END_VAR
IF NOT pInternal^ THEN
	pInternal^			:= TRUE;
	pPublic^			:= TRUE;	
ELSIF NOT pPublic^ THEN
	pInternal^			:= FALSE;
	pAcknowledgement^	:= TRUE;
END_IF
END_METHOD

END_FUNCTION_BLOCK

// ---- Machine System/PRGs/CAM_CNC/CNC/PRG_ManualModeVirtualHBA.TcPOU
PROGRAM PRG_ManualModeVirtualHBA
VAR_INPUT
	nChanIdx						: UDINT;			(* Number of channel *)
	bEnable 					: BOOL;
END_VAR

VAR_IN_OUT
	stManualModeParameter 		: ST_ManualModeParameter;
	stManualModeControlElements : ST_ManualModeControlElements;
END_VAR

VAR
	RTRIG_RapidKey : R_TRIG;
END_VAR

stManualModeParameter.stChannelParameter.nChanIdx							:= 0;       (* Kanal 1 *)
stManualModeParameter.stChannelParameter.nInc					:= 1;

(*  Manual Type Selection*)
IF (stVirtualHBA[nChanIdx].KeyHW.bKey) THEN
	stManualModeParameter.stChannelParameter.eManualType := 1;
END_IF

IF (stVirtualHBA[nChanIdx].KeyTipp.bKey) THEN
	stManualModeParameter.stChannelParameter.eManualType := 2;
END_IF

IF (stVirtualHBA[nChanIdx].KeyJog.bKey) THEN
	stManualModeParameter.stChannelParameter.eManualType := 3;
END_IF

IF (stVirtualHBA[nChanIdx].KeyJS.bKey) THEN
	stManualModeParameter.stChannelParameter.eManualType := 4;
END_IF

stVirtualHBA[nChanIdx].KeyTipp.bLED 	:= FALSE;
stVirtualHBA[nChanIdx].KeyJog.bLED 	:= FALSE;
stVirtualHBA[nChanIdx].KeyHW.bLED 	:= FALSE;
stVirtualHBA[nChanIdx].KeyJS.bLED 	:= FALSE;

IF NOT bEnable OR stVirtualHBA[nChanIdx].nLogAxisId = 0 THEN
	RETURN;
END_IF




CASE CNCSystem.Channel[nChanIdx].ActMode OF

HLI_IMCM_MANUAL_MODE:
	CASE stManualModeParameter.stChannelParameter.eManualType OF
		1: stVirtualHBA[nChanIdx].KeyHW.bLED 		:= TRUE;
		2: stVirtualHBA[nChanIdx].KeyTipp.bLED 	:= TRUE;
		3: stVirtualHBA[nChanIdx].KeyJog.bLED 		:= TRUE;
		4: stVirtualHBA[nChanIdx].KeyJS.bLED 		:= TRUE;
	END_CASE
END_CASE

(*  AxisID Selection*)
stManualModeParameter.stAxisParameter.stControlUnit[0].nLogAxisNr := UINT_TO_INT(stVirtualHBA[nChanIdx].nLogAxisId);

(* Handwheel Inc *)
stManualModeControlElements.nHandwheelInc[0] := stVirtualHBA[nChanIdx].nHandwheelInc;

(* Jog Increments *)
stManualModeParameter.stChannelParameter.nInc := stVirtualHBA[nChanIdx].nJogInc;

(* Axis Speed *)
stManualModeParameter.stAxisParameter.stControlUnit[0].nSpeed := stVirtualHBA[nChanIdx].nSpeed;
stManualModeParameter.stAxisParameter.stControlUnit[1].nSpeed := stVirtualHBA[nChanIdx].nSpeed;

(* Manual Mode initialization Parameter *)
stManualModeParameter.stChannelParameter.strInitParameter := stVirtualHBA[nChanIdx].strInitParameter;

(* Joystick *)
stManualModeControlElements.stControlJoystickValue[0] := stVirtualHBA[nChanIdx].nJoystickValue1;
stManualModeControlElements.stControlJoystickValue[1] := stVirtualHBA[nChanIdx].nJoystickValue2;

IF (stManualModeParameter.stChannelParameter.eManualType = 4) THEN
	stManualModeParameter.stAxisParameter.stControlUnit[0].nLogAxisNr := 1;
	stManualModeParameter.stAxisParameter.stControlUnit[1].nLogAxisNr := 2;
ELSE
	stManualModeParameter.stAxisParameter.stControlUnit[1].nLogAxisNr := 0;
END_IF


(* Handwheel and Joystick settings *)
stManualModeParameter.stChannelParameter.nHandwheelResolution 		:= stVirtualHBA[nChanIdx].nHandwheelResolution;
stManualModeParameter.stJoystickParameter.AnalogValueZeroDeadBand 	:= stVirtualHBA[nChanIdx].nAnalogValueZeroDeadBand;
stManualModeParameter.stJoystickParameter.AnalogValueMax 			:= stVirtualHBA[nChanIdx].nAnalogValueMax;
stManualModeParameter.stJoystickParameter.AnalogValueMin 			:= stVirtualHBA[nChanIdx].nAnalogValueMin;

(* Direction key_s *)				
stManualModeControlElements.stControlKeys[0].bKeyNeg := stVirtualHBA[nChanIdx].KeyNeg.bKey;
stManualModeControlElements.stControlKeys[0].bKeyPos := stVirtualHBA[nChanIdx].KeyPos.bKey;

(* Rapid key *)
RTRIG_RapidKey(CLK:= stVirtualHBA[nChanIdx].KeyRapid.bKey);

IF RTRIG_RapidKey.Q AND NOT stManualModeControlElements.stControlKeys[0].bKeyRapid THEN
	stManualModeControlElements.stControlKeys[1].bKeyRapid := TRUE;
ELSIF RTRIG_RapidKey.Q AND stManualModeControlElements.stControlKeys[0].bKeyRapid THEN
	  stManualModeControlElements.stControlKeys[1].bKeyRapid := FALSE;
END_IF

stVirtualHBA[nChanIdx].KeyRapid.bLED := stManualModeControlElements.stControlKeys[0].bKeyRapid AND
								(CNCSystem.Channel[nChanIdx].ActMode = HLI_IMCM_MANUAL_MODE);

stVirtualHBA[nChanIdx].KeyNeg.bLED := stManualModeControlElements.stControlKeys[0].bKeyNeg;
stVirtualHBA[nChanIdx].KeyPos.bLED := stManualModeControlElements.stControlKeys[0].bKeyPos;


(* Status *)
stVirtualHBA[nChanIdx].nStatusManualType := stManualModeParameter.stChannelParameter.eManualType;

END_PROGRAM

// ---- Machine System/PRGs/CAM_CNC/CNC/myPlcAxis.TcPOU
PROGRAM myPlcAxis
VAR
	fbAxis_X 					: FB_CNCAxis; 
	fbMoveAbsolute 				: MC_MOVEAbsolute;	
	fbSetOverride 				: MC_SetOverride;	
	fbStop						: MC_Halt;	
	bStop 						: BOOL;
	bSetRefPos: BOOL;
	bExecuteMoveAbsolute: BOOL;
	rXposReq: LREAL;
	rXvelReq: LREAL := 1000;
	rtAxPlcMode: R_TRIG;
	bEnterAxPlcMode: BOOL;
	nCase: INT;
	fbCSV: FB_CSV_RECIPE;
	arrCSVData : ARRAY [0..1, 0..MAX_CSV_ROWS] OF STRING(MAX_CSV_FIELD_LENGTH);
	bReadCsv : BOOL;
	bWriteCsv : BOOL;
	fbMoveRel: MC_MoveRelative;
	bMoveRel : BOOL;
	fbHome: MC_Home;
	bHomeExe : BOOL;
	bHomeSw : BOOL;
	fbPower: MC_Power;
	bEnable : bool;
END_VAR

// example of moving a CNC axis that is part of a channel with PLC Move Absolute.  
// Note, this is absolute position of axis, no CNC offsets are applied!!!
// When entering this "mode", the channel needs to be set to Select, then Ready before executing PLC moves
// axis must be homed before PLC moves are allowed
// When leaving this "mode", the channel needs to be Reset, or #CHANNEL INIT[CMDPOS] needs called from MDI or Auto in order for the position commands to be correct.
// this code requires Tc2_CncBase and Tc2_CncPlcOpenP1 libraries to be added
// Axis needs to have this parameter added "Kenngr.enable_single_axis    1    (P-AXIS-00457".  This allows the axis to be PLC controlled

// only need to call this next FUN if the axis is not homed or not using abs encoders.  Must be homed for PLC axis to work.
HLI3_SetAxisReferencePosition(bSetRefpos:= bSetRefPos, nHliAxisIdx:= 2);  // X axis example


rtAxPlcMode(CLK:= bEnterAxPlcMode, Q=> );
IF rtAxPlcMode.Q AND fbAxis_X.stStatus.bHomingDone AND fbAxis_X.stStatus.bIsEnabled THEN
	nCase := 10;
END_IF

CASE nCase OF
	10: // channel 0 to select, then wait for acutal state to be select
		PLCMachineMode[0].Select := TRUE;
		IF PRG_CNCChannelHandler.CNCChannel[0].currentstate = 2 THEN
			nCase := 20;
		END_IF
		
	20: // channel 0 to ready, then wait for acutal state to be ready
		PLCMachineMode[0].Ready := TRUE;
		IF PRG_CNCChannelHandler.CNCChannel[0].currentstate = 3 THEN
			nCase := 0;
		END_IF
END_CASE

fbHome(
	Axis:= g_array_axis_ref[CNCSystem.LogAxisNo[3].nHliAxisIdx], 
	Execute:= bHomeExe, 
	CamSignal:= bHomeSw, 
	Done=> , 
	CommandAborted=> , 
	Error=> , 
	ErrorID=> );
(*	
fbPower(
	Axis:= g_array_axis_ref[CNCSystem.LogAxisNo[3].nHliAxisIdx], 
	Enable:= bEnable, 
	Enable_Positive:= 1, 
	Enable_Negative:= 1, 
	PowerDefaultState:= , 
	DriveEnabled=> , 
	DriveReady=> , 
	PowerState=> , 
	Status=> , 
	Error=> , 
	ErrorID=> );
*)
fbAxis_X(
	nLogAxisNo:= 3, 
	bEnable:= PLCAxisEnable, 
	bCalibrationCam:=, 
	bSetRefOffset:= , 
	fRefOffset:= , 
	bFeedhold:= ,		 
	stStatus=> );
		
fbSetOverride(
	Axis:= g_array_axis_ref[CNCSystem.LogAxisNo[3].nHliAxisIdx],  
	Enable:= bEnterAxPlcMode, //TRUE, 
	VelFactor:= 1, 
	VelFactorMaxShift:=1 , 
	Enabled=> , 
	Error=> , 
	ErrorID=> );

		
fbMoveAbsolute(
	Axis:= g_array_axis_ref[CNCSystem.LogAxisNo[3].nHliAxisIdx], 
	Execute:= bExecuteMoveAbsolute AND (PRG_CNCChannelHandler.CNCChannel[0].currentstate = 3), 
	Position:= rXposReq*10000, 
	Velocity:= rXvelReq * 16.6666, 
	Acceleration:= 200, // adj per application
	Deceleration:= 200, // adj per application
	Jerk:= 500,         // adj per application
	Direction:= , 
	Done=> , 
	CommandAborted=> , 
	Error=> , 
	ErrorID=> );
	
fbMoveRel(
	Axis:= g_array_axis_ref[CNCSystem.LogAxisNo[3].nHliAxisIdx], 
	Execute:= bMoveRel, 
	Distance:= 12.0*10000, 
	Velocity:= rXvelReq * 16.6666, 
	Acceleration:= 200, 
	Deceleration:= 200, 
	Jerk:= 500, 
	Done=> , 
	CommandAborted=> , 
	Error=> , 
	ErrorID=> );
 
fbStop(
	Axis:= g_array_axis_ref[CNCSystem.LogAxisNo[3].nHliAxisIdx], 
	Execute:= bStop, 
	Deceleration:= 1000, 
	Jerk:= , 
	Done=> , 
	CommandAborted=> , 
	Error=> , 
	ErrorID=> );		
	
	
PRG_CNCChannelHandler.CNCChannel[0].currentMode;

Tc3_CNC.GLOBAL_CNC.cncsystem.channel[0].ActMode;

fbCSV(
	bReadCSV:= bReadCsv, 
	bWriteCSV:= bWriteCsv, 
	sFile:= 'C:\Temp\bacjunk_Units.csv', 
	sDelimeter:= ',', 
	bBusy=> , 
	bErr=> , 
	bReadingDone=> , 
	bWritingDone=> , 
	arrCSVData:= arrCSVData);

END_PROGRAM

// ---- Machine System/PRGs/CSV/FB_CSV_RECIPE.TcPOU
FUNCTION_BLOCK FB_CSV_RECIPE
VAR_INPUT
	bReadCSV : BOOL;
	bWriteCSV  : BOOL;
	sFile : STRING(255);
	sDelimeter : STRING;
END_VAR
VAR_OUTPUT
	bBusy : BOOL;
	bErr : BOOL;
	bReadingDone : BOOL;
	bWritingDone : BOOL;
END_VAR
VAR
	fbFileOpen: FB_FileOpen;
	eOpenMode : UDINT;
	bOpen : BOOL;
	fbFileClose: FB_FileClose;
	bClose: BOOL;
	fbFilePuts: FB_FilePuts;
	bWriteLine: BOOL;
	fbFileGets: FB_FileGets;
	bGetLine: BOOL;
	sLine2Write: T_MaxString;
	sLastLineRead: T_MaxString;
	hFile: UINT;
	i: UDINT;
	rtRead: R_TRIG;
	rtWrite: R_TRIG;
	step: INT;
	n: UDINT;
	iCommaPos: INT;
	sColumn: ARRAY [0..MAX_CSV_COLUMNS] OF STRING(MAX_CSV_FIELD_LENGTH);
	iStringLen: INT;
	bWritingBusy : BOOL;
	bReadingBusy : BOOL;
	sTempString: STRING(MAX_CSV_FIELD_LENGTH);
END_VAR

VAR_IN_OUT
	arrCSVData : ARRAY [0..1, 0..MAX_CSV_ROWS] OF STRING(MAX_CSV_FIELD_LENGTH);
END_VAR

(* this code requires that these global constants are declared......as "VAR_GLOBAL CONSTANT"
VAR_GLOBAL CONSTANT
	MAX_CSV_ROWS 			: UDINT := 100;
	MAX_CSV_COLUMNS 		: UDINT := 5;
	MAX_CSV_FIELD_LENGTH	: UDINT := 100;
END_VAR
*)
IF bReadingDone AND NOT bReadCSV THEN
	bReadingDone := FALSE;
END_IF
IF bWritingDone AND NOT bWriteCSV THEN
	bWritingDone := FALSE;
END_IF

rtRead(CLK:= bReadCSV, Q=> );
rtWrite(CLK:= bWriteCSV, Q=> );

IF rtRead.Q AND NOT bWriteCSV THEN
	bReadingBusy := TRUE;
	step := 10;
END_IF

IF rtWrite.Q AND NOT bReadCSV THEN
	bWritingBusy := TRUE;
	step := 110;
END_IF


	CASE step OF
		10: (* set to init values *)
			bOpen := FALSE; bClose := FALSE; bWriteLine := FALSE; bGetLine := FALSE; bErr := FALSE; bReadingDone := FALSE; bWritingDone := FALSE;
			bBusy := TRUE;
			n := 0;
			step := 20;

		20:	(* set mode for reading *)
			eOpenMode := FOPEN_MODEAPPEND OR FOPEN_MODEPLUS;
			bOpen := TRUE;
			IF fbFileOpen.bBusy THEN
				bOpen := FALSE;
				step := 30;
			END_IF
		30:
			IF NOT fbFileOpen.bBusy THEN
				IF NOT fbFileOpen.bError THEN
					step := 40;
				ELSE
					step := 999;
				END_IF
			END_IF
		40:
			bGetLine := TRUE;
			IF fbFileGets.bBusy THEN
				bGetLine := FALSE;
				step := 50;
			END_IF
		50:
			IF NOT fbFileGets.bBusy THEN
				IF NOT fbFileGets.bError THEN
					step := 60;
				ELSE
					step := 999;
				END_IF
			END_IF
		60:
			A_ParseCSV();
			FOR i := 0 TO MAX_CSV_COLUMNS BY 1 DO
				arrCSVData[i,n] := sColumn[i];
			END_FOR
			n := n + 1;
			step := 70;
		70:
			IF n >= MAX_CSV_ROWS THEN
				step := 200;
			ELSE
				step := 40;
			END_IF


		(* writing *)
		110:
			bOpen := FALSE; bClose := FALSE; bWriteLine := FALSE; bGetLine := FALSE; bErr := FALSE;
			bBusy := TRUE;
			n := 0;
			step := 120;

		120:
			eOpenMode := FOPEN_MODEWRITE;
			bOpen := TRUE;
			IF fbFileOpen.bBusy THEN
				bOpen := FALSE;
				step := 130;
			END_IF
		130:
			IF NOT fbFileOpen.bBusy THEN
				IF NOT fbFileOpen.bError THEN
					step := 140;
				ELSE
					step := 999;
				END_IF
			END_IF
		140:
			sLine2Write := CONCAT(arrCSVData[0,n],sDelimeter);
			FOR i := 1 TO MAX_CSV_COLUMNS-1 BY 1 DO
				sLine2Write := CONCAT(sLine2Write,arrCSVData[i,n]);
				sLine2Write := CONCAT(sLine2Write,sDelimeter);
			END_FOR
			sLine2Write := CONCAT(sLine2Write,arrCSVData[MAX_CSV_COLUMNS,n]);
			sLine2Write := CONCAT(sLine2Write, '$N');
			bWriteLine := TRUE;
			step := 150;
		150:
			IF fbFilePuts.bBusy THEN
				bWriteLine := FALSE;
				step := 160;
			END_IF
		160:
			IF NOT fbFilePuts.bBusy THEN
				IF NOT fbFilePuts.bError THEN
					step := 170;
				ELSE
					step := 999;
				END_IF
			END_IF
		170:
			n := n + 1;
			IF n >= MAX_CSV_ROWS THEN
				step := 200;
			ELSE
				step := 140;
			END_IF


		(* close file *)
		200:
			bClose := TRUE;
			IF fbFileClose.bBusy THEN
				bClose := FALSE;
				step := 210;
			END_IF
		210:
			IF NOT fbFileClose.bError THEN
				IF bWritingBusy THEN
					bWritingBusy := FALSE;
					bWritingDone := TRUE;
				ELSIF bReadingBusy THEN
					bReadingBusy := FALSE;
					bReadingDone := TRUE;
				END_IF
				bBusy := FALSE;
				step := 0;
			END_IF

		999:
			bOpen := FALSE;  bWriteLine := FALSE; bGetLine := FALSE; bReadingDone := FALSE; bWritingDone := FALSE; bBusy := FALSE;
			bErr := TRUE;
			bClose := TRUE;
	END_CASE


fbFileOpen(
	sNetId:= ,
	sPathName:= sFile,
	nMode:= eOpenMode,
	ePath:= ,
	bExecute:= bOpen,
	tTimeout:= ,
	bBusy=> ,
	bError=> ,
	nErrId=> ,
	hFile=> hFile);

fbFilePuts(
	sNetId:= ,
	hFile:= hFile,
	sLine:= sLine2Write,
	bExecute:= bWriteLine,
	tTimeout:= ,
	bBusy=> ,
	bError=> ,
	nErrId=> );

fbFileGets(
	sNetId:= ,
	hFile:= hFile,
	bExecute:= bGetLine,
	tTimeout:= ,
	bBusy=> ,
	bError=> ,
	nErrId=> ,
	sLine=> sLastLineRead,
	bEOF=> );

fbFileClose(
	sNetId:= ,
	hFile:= hFile,
	bExecute:= bClose,
	tTimeout:= ,
	bBusy=> ,
	bError=> ,
	nErrId=> );

IF fbFileOpen.bError OR fbFilePuts.bError OR fbFileGets.bError OR fbFileClose.bError THEN
	bErr := TRUE;
	bOpen := FALSE;  bWriteLine := FALSE; bGetLine := FALSE; bReadingDone := FALSE; bWritingDone := FALSE; bBusy := FALSE;
	IF hFile <> 0 THEN
		bClose := TRUE;
	END_IF
END_IF

ACTION A_ParseCSV:
sTempString := sLastLineRead;
 
FOR i := 0 TO MAX_CSV_COLUMNS BY 1 DO
                                iCommaPos:= FIND(STR1:= sTempString, STR2:= sDelimeter);
                                iStringLen := LEN(STR:= sTempString);
                                sColumn[i] := MID(STR:= sTempString, LEN:= iCommaPos-1, POS:= 1);
                                sTempString := MID(STR:= sTempString, LEN:= iStringLen - iCommaPos, POS:= iCommaPos+1);
END_FOR
END_ACTION

END_FUNCTION_BLOCK

// ---- Machine System/PRGs/CAM_CNC/CNC/myPlcAxis_1.TcPOU
PROGRAM myPlcAxis_1
VAR
	fbAxis_X 					:  FB_CNCAxis; 
	fbMoveAbsolute 				: MC_MOVEAbsolute;	
	fbMoveafterTipTouch			: MC_MoveSuperImposed;
	
	fbTouchProbe				: MC_TouchProbe;
	fbMoveIncrement				: MC_MOVERelative; 
	 
	
	fbSetOverride 				: MC_SetOverride;	
	fbStop						: MC_Halt;	
	bStop 						: BOOL;
	bSetRefPos: BOOL;
	bExecuteMoveAbsolute: BOOL;
	rXposReq: LREAL;
	rXvelReq: LREAL := 1000;
	rtAxPlcMode: R_TRIG;
	bEnterAxPlcMode: BOOL;
	nCase: INT;
	
	startZCal: BOOL;
	rZposReq: INT;
	rZvelReq: INT;
	
	tipTouch : BOOL; 
	CalibrateHSS: BOOL;
	Zat12MM: BOOL;
	ZatTipTouch: BOOL := FALSE;
	Failedtoreach12mm: BOOL;
	travelto100mmDone: BOOL;
	
	// Fbstop
	PlCmoveStopped: BOOL;
	PLCstopAborted: BOOL;
	PLCstopError: BOOL;
	
	// Absolute
	travelto100mmAborted: BOOL;
	travelto100mmError: BOOL;
	// Increment
	ErrortoReach12mm: BOOL;
	
//	ZmovetotipTouch : ZaxisAbsolute;
//	Zmoveto12MM		: HSSCalibrationat12MM;
	ErrId: WORD;
	bExecuteMoveIncrement: BOOL;
	rZ_ActPos: LREAL;
	ZPosatTipTouch: LREAL;
	Zto12MM: LREAL;
	CalTmr : TON;
	wHS_DigInputs: WORD;
	nZCalStep : INT;
	rtZcal: R_TRIG;
END_VAR


// HSS Calibration Variable Init
tipTouch := wHS_DigInputs.1;			// Tip touch from the FC2D cutting head
//OUT.wHS_DigOutputs.0 := CalibrateHSS; 		// Set Calibrate HSS output

rZ_ActPos := HLI3_GetActualAxisPos(nHliAxisIdx:= 2) * 0.0001;

// Z-axis absolute and increment move setup
HLI3_SetAxisReferencePosition(bSetRefpos:= bSetRefPos, nHliAxisIdx:= 2);	// Z axis

rtAxPlcMode(CLK:= bEnterAxPlcMode, Q=> );
IF rtAxPlcMode.Q AND fbAxis_X.stStatus.bHomingDone AND fbAxis_X.stStatus.bIsEnabled THEN
	nCase := 10;
END_IF

CASE nCase OF
	10: // channel 0 to select, then wait for acutal state to be select
		PLCMachineMode[0].Select := TRUE;
		IF PRG_CNCChannelHandler.CNCChannel[0].currentstate = 2 THEN
			nCase := 20;
		END_IF
		
	20: // channel 0 to ready, then wait for acutal state to be ready
		PLCMachineMode[0].Ready := TRUE;
		IF PRG_CNCChannelHandler.CNCChannel[0].currentstate = 3 THEN
			nCase := 100;
		END_IF
END_CASE


	
rtZcal(CLK:= startZCal, Q=> );			
IF rtZcal.Q THEN	
	startZCal := FALSE;
	bEnterAxPlcMode := TRUE;
	nZcalStep := 10;
END_IF
		
CASE nZCalStep OF
	10:
		IF nCase = 100 THEN
			IF NOT tipTouch THEN
				// Travel to negative limit until tip touch
				bExecuteMoveAbsolute := TRUE;
				nZcalStep := 20;
				//ZatTipTouch := TRUE;	
			END_IF
		END_IF
		
	20:
		IF tipTouch THEN
			bExecuteMoveAbsolute := FALSE;
			bExecuteMoveIncrement := TRUE;
			nZcalStep := 30;
		ELSIF fbMoveAbsolute.Done THEN
			bExecuteMoveAbsolute := FALSE;
			nZcalStep := 999;
		END_IF
	30:
		CalibrateHSS := TRUE;
		IF CalTmr.Q THEN
			CalibrateHSS := FALSE;
			nZCalStep := 40;
		END_IF 
		
	40:
		IF fbMoveIncrement.Done THEN
			bExecuteMoveAbsolute := FALSE;
			bExecuteMoveIncrement := FALSE;
			bEnterAxPlcMode := FALSE;
			nZCalStep := 100;
		END_IF
		
END_CASE
		
CalTmr (IN := CalibrateHSS, PT := T#0.1S);		
		
fbAxis_X(
	nLogAxisNo:= 3, 
	bEnable:= PLCAxisEnable, 
	bCalibrationCam:=, 
	bSetRefOffset:= , 
	fRefOffset:= , 
	bFeedhold:= ,		 
	stStatus=> );


fbSetOverride(
	Axis:= g_array_axis_ref[CNCSystem.LogAxisNo[3].nHliAxisIdx],  
	Enable:= bEnterAxPlcMode, 
	VelFactor:= 1, 
	VelFactorMaxShift := 1 , 
	Enabled=> , 
	Error=> , 
	ErrorID=> );

// Absolute
fbMoveAbsolute(
	Axis:= g_array_axis_ref[CNCSystem.LogAxisNo[3].nHliAxisIdx], 
	Execute:= bExecuteMoveAbsolute AND (PRG_CNCChannelHandler.CNCChannel[0].currentstate = 3), 
	Position:= -40*10000, 
	Velocity:= 150 * 16.6666, 
	Acceleration:= 200, // adj per application
	Deceleration:= 200, // adj per application
	Jerk:= 500,         // adj per application
	Direction:= , 
	Done=> travelto100mmDone, 
	CommandAborted=> travelto100mmAborted, 
	Error=> travelto100mmError, 
	ErrorID=> ErrId);


// Increment
fbMoveIncrement(
	Axis:= g_array_axis_ref[CNCSystem.LogAxisNo[3].nHliAxisIdx], 
	Execute:= bExecuteMoveIncrement AND (PRG_CNCChannelHandler.CNCChannel[0].currentstate = 3),
	Distance:= 12*10000, 
	Velocity := 150 * 16.6666, 
	Acceleration:= 200, // adj per application
	Deceleration:= 200, // adj per application
	Jerk:= 500,         // adj per application
	Done=> Zat12MM, 
	CommandAborted=> Failedtoreach12mm, 
	Error=> ErrortoReach12mm, 
	ErrorID=> ErrId);

END_PROGRAM

// ---- Machine System/PRGs/CAM_CNC/CNC/myPRG_AxisHomeSwitches.TcPOU
PROGRAM myPRG_AxisHomeSwitches
VAR
	
	i: USINT;
	xHomed_X: BOOL;
	xHomed_Y: BOOL;
	xHomed_Z: BOOL;
END_VAR


HLI3_SetAxisReferenceCam(nHliAxisIdx := 0, bReferenceCam := bXHomeSwitch);
HLI3_SetAxisReferenceCam(nHliAxisIdx := 1, bReferenceCam := bYHomeSwitch);
HLI3_SetAxisReferenceCam(nHliAxisIdx := 2, bReferenceCam := bZHomeSwitch);

// Below sets all axis positions to zero and sets "homed" flag
//HLI3_SetAxisReferencePosition(bSetRefpos:= bSet, nHliAxisIdx:= 0); // cannot be done in manual mode
//HLI3_SetAxisReferencePosition(bSetRefpos:= bSet, nHliAxisIdx:= 1); // cannot be done in manual mode
//HLI3_SetAxisReferencePosition(bSetRefpos:= bSet, nHliAxisIdx:= 2); // cannot be done in manual mode

//Axis Home Status i.e. is the axis home
xHomed_X := gpAx[0]^.lr_state.homing_done_r;
xHomed_Y := gpAx[1]^.lr_state.homing_done_r;
xHomed_Z := gpAx[2]^.lr_state.homing_done_r;

END_PROGRAM

// ---- Machine System/PRGs/CAM_CNC/CNC/myPRG_CNCManualMode_1.TcPOU
PROGRAM myPRG_CNCManualMode_1
VAR
	fbUintUdInt: FB_Uint_Udint;
	nHandwheelSmall AT %I*: UINT;		(* increments for handwheel (e.g. EL5101   *)
	nHandwheelPreset AT %Q* : UINT := 32767;
	nHandWheelBig: UDINT;
	bZeroHandWheel AT %Q* : BOOL;
	
	rtHandWheelEnable: R_TRIG;
	nCase: INT;
	bHandWheelEnabled: BOOL;
	ftHandWheelEnabled: F_TRIG;
	nHwCounts : UINT;
	nLastCounts : UINT;
	tmrHandWheelOnDelay: TON;
	tmrJogX: TON;
	tmrJogY: TON;
	tmrJogZ: TON;
END_VAR

// edited to for use of physical push buttons instead of touch screen buttons
//FOR i := 0 TO MAX_USED_CHANNEL_IDX DO

	IF (HLI3_CheckChannelValid(0)) THEN

		stManualModeParameter[0].stChannelParameter.nChanIdx := 0;       (* Channel 1 *)
		stManualModeParameter[0].stChannelParameter.nInc := PLCMachineMode[0].ManualMode.nInc;
		stManualModeParameter[0].stChannelParameter.eManualType := UINT_TO_INT(PLCMachineMode[0].ManualMode.nManualTyp);
		stManualModeParameter[0].stChannelParameter.nHandwheelResolution := PLCMachineMode[0].ManualMode.nHwResolution;    (* 0.1 µm /rev (from HMI) *)
		stManualModeParameter[0].stAxisParameter.stControlUnit[0].nLogAxisNr := PLCMachineMode[0].ManualMode.nLogAxisNumber;   (* Log. Achs Nummer *)
		IF stManualModeParameter[0].stAxisParameter.stControlUnit[0].nLogAxisNr = 0 THEN
			stManualModeParameter[0].stAxisParameter.stControlUnit[0].nLogAxisNr := gpCh[0]^.bahn_state.coord_r[0].log_achs_nr_r;
			PLCMachineMode[0].ManualMode.nLogAxisNumber := gpCh[0]^.bahn_state.coord_r[0].log_achs_nr_r;
		END_IF
		stManualModeParameter[0].stAxisParameter.stControlUnit[0].nSpeed := LREAL_TO_UINT(PLCMachineMode[0].ManualMode.nSpeed * 16.666);
		stManualModeControlElements[0].stControlKeys[0].bKeyRapid := PLCMachineMode[0].ManualMode.bKeyRapid := bRapidPB;
		//stManualModeControlElements[0].nHandwheelInc
		
  END_IF
//END_FOR


(* edited for handwheel axis selection *)
bHandWheelEnabled := bMpgSelect1 OR bMpgSelect10 OR bMpgSelect100;
rtHandWheelEnable(CLK:= bHandWheelEnabled);
IF rtHandWheelEnable.Q THEN
	nCase := 10;
END_IF
ftHandWheelEnabled(CLK:= bHandWheelEnabled, Q=> );
IF ftHandWheelEnabled.Q THEN
	PLCMachineMode[1].ManualMode.nManualTyp := 2;
	nCase := 0;
END_IF
tmrHandWheelOnDelay(IN:= bHandWheelEnabled, PT:= t#150ms, Q=> , ET=> );
CASE nCase OF
	10:
		IF tmrHandWheelOnDelay.Q THEN
			nCase := 20;
		END_IF
		
	20:
		bZeroHandWheel := true;
		IF nHandwheelSmall = 32767 THEN
			nLastCounts := nHandwheelSmall;
			bZeroHandWheel := false;
			nCase := 30;
		END_IF
		
	30:
		IF nLastCounts <> nHandwheelSmall THEN
			nHwCounts := nHwCounts + (nHandwheelSmall - nLastCounts);
			nLastCounts := nHandwheelSmall;
		END_IF
		PLCMachineMode[0].ManualMode.nManualTyp := 1;
		IF bMpgSelectX THEN
			PLCMachineMode[0].ManualMode.nLogAxisNumber := 1;
		ELSIF bMpgSelectY THEN
			PLCMachineMode[0].ManualMode.nLogAxisNumber := 2;
		ELSIF bMpgSelectZ THEN
			PLCMachineMode[0].ManualMode.nLogAxisNumber := 3;
		ELSE
			PLCMachineMode[0].ManualMode.nLogAxisNumber := -1;
		END_IF
		
		IF bMpgSelect1 THEN
			PLCMachineMode[0].ManualMode.nHwResolution := 1;
		ELSIF bMpgSelect10 THEN
			PLCMachineMode[0].ManualMode.nHwResolution := 10;
		ELSIF bMpgSelect100 THEN
			PLCMachineMode[0].ManualMode.nHwResolution := 100;
		END_IF
	
END_CASE
fbUintUdInt(nInSmall := nHwCounts, nBig := nHandWheelBig);
stManualModeControlElements[0].nHandwheelInc[0] :=  nHandWheelBig *100;

(* edited for manual jog buttons *)

IF bJogRevX OR bJogFwdX THEN
	PLCMachineMode[0].ManualMode.nLogAxisNumber := 1;
ELSIF bJogRevY OR bJogFwdY THEN
	PLCMachineMode[0].ManualMode.nLogAxisNumber := 2;
ELSIF bJogRevZ OR bJogFwdZ THEN
	PLCMachineMode[0].ManualMode.nLogAxisNumber := 3;
END_IF

tmrJogX(IN:= bJogRevX OR bJogFwdX, PT:= T#80MS);
tmrJogY(IN:= bJogRevY OR bJogFwdY, PT:= T#80MS);
tmrJogZ(IN:= bJogRevZ OR bJogFwdZ, PT:= T#80MS);
IF stManualModeParameter[0].stAxisParameter.stControlUnit[0].nLogAxisNr = 1 AND tmrJogX.Q THEN
	stManualModeControlElements[0].stControlKeys[0].bKeyNeg	:= PLCMachineMode[0].ManualMode.bKeyNeg := bJogRevX;
	stManualModeControlElements[0].stControlKeys[0].bKeyPos	:= PLCMachineMode[0].ManualMode.bKeyPos := bJogFwdX;
ELSIF stManualModeParameter[0].stAxisParameter.stControlUnit[0].nLogAxisNr = 2 AND tmrJogY.Q THEN
	stManualModeControlElements[0].stControlKeys[0].bKeyNeg	:= PLCMachineMode[0].ManualMode.bKeyNeg := bJogRevY;
	stManualModeControlElements[0].stControlKeys[0].bKeyPos	:= PLCMachineMode[0].ManualMode.bKeyPos := bJogFwdY;
ELSIF stManualModeParameter[0].stAxisParameter.stControlUnit[0].nLogAxisNr = 3 AND tmrJogZ.Q THEN
	stManualModeControlElements[0].stControlKeys[0].bKeyNeg	:= PLCMachineMode[0].ManualMode.bKeyNeg := bJogRevZ;
	stManualModeControlElements[0].stControlKeys[0].bKeyPos	:= PLCMachineMode[0].ManualMode.bKeyPos := bJogFwdZ;
ELSE
	stManualModeControlElements[0].stControlKeys[0].bKeyNeg	:= PLCMachineMode[0].ManualMode.bKeyNeg := FALSE;
	stManualModeControlElements[0].stControlKeys[0].bKeyPos	:= PLCMachineMode[0].ManualMode.bKeyPos := FALSE;
END_IF

END_PROGRAM

// ---- Machine System/PRGs/CAM_CNC/CNC/PRG_SetAxisOffsets.TcPOU
PROGRAM PRG_SetAxisOffsets
VAR
	fbSetAxisZero_X1: FB_SetAxisZero;
	fbSetAxisZero_X2: FB_SetAxisZero;
	fbSetAxisZero_Y: FB_SetAxisZero;
	bSetZeroX : BOOL;
	bSetZeroY : BOOL;
END_VAR

//These need declared.....
(*VAR_GLOBAL PERSISTENT
	rX1Offset: LREAL;
	rX2Offset: LREAL;
	rYOffset: LREAL;
END_VAR*)

fbSetAxisZero_X1(
	nHliAxisIdx:= 0, 
	bExecute:= bSetZeroX, 
	bWriteOnStart:= TRUE,
	rOffset:= rX1Offset, 
	bBusy=> , 
	bDone=> , 
	bError=> );

fbSetAxisZero_X2(
	nHliAxisIdx:= 3, 
	bExecute:= bSetZeroX, 
	bWriteOnStart:= TRUE,
	rOffset:= rX2Offset, 
	bBusy=> , 
	bDone=> , 
	bError=> );

fbSetAxisZero_Y(
	nHliAxisIdx:= 1, 
	bExecute:= bSetZeroY, 
	bWriteOnStart:= TRUE,
	rOffset:= rYOffset, 
	bBusy=> , 
	bDone=> , 
	bError=> );

END_PROGRAM

// ---- Machine System/PRGs/CAM_CNC/myCNC_Call_BogieIndex.TcPOU
PROGRAM myCNC_Call_BogieIndex
VAR
END_VAR

END_PROGRAM

// ---- Machine System/PRGs/CAM_CNC/myCNC_Call_Place.TcPOU
PROGRAM myCNC_Call_Place
VAR
END_VAR

END_PROGRAM

// ---- Machine System/PRGs/CAM_CNC/myCNC_Call_Roll.TcPOU
PROGRAM myCNC_Call_Roll
VAR
END_VAR

END_PROGRAM

// ---- Machine System/PRGs/CAM_CNC/myCNC_Call_Spray.TcPOU
PROGRAM myCNC_Call_Spray
VAR
	ncase : INT;
	
	JobCase 	: INT;
	SD1State 	: INT; //0:Pickup, 1:SprayA, 2: rollA, 3:placeA, 4:cureA, 5:SprayB, 6:RollB, 7:PlaceB, 8:CureB, 9:SetDown, 10:Traveling
	SD2State 	: INT;	//0:Pickup, 1:SprayA, 2: rollA, 3:placeA, 4:cureA, 5:SprayB, 6:RollB, 7:PlaceB, 8:CureB, 9:SetDown, 10:Traveling
	
	RailPriority	: INT;
	SprayQue	: ARRAY[0..20] OF STRING;
	
	WX1SprayJob		: MoldJob;
	WX2SprayJob		: MoldJob;
	WX3SprayJob		: MoldJob;
	WX4SprayJob		: MoldJob;
END_VAR

(* adjust for wxjob and start calls in the JobCase instead of Ncase 10-25-22
IF SectionAKey AND PRG_CNCChannelHandler.CNCChannel[0].currentmode = 4 THEN
	SectionAKey := FALSE;
	nCase := 10;
END_IF

*)
//add job to spray que from Job Que
	//set priority to SD1 or SD2 based on FIFO skip adding to que and just change job priority
	// If SD1 complete then RailPriority = 2
//check which rail is prio and which job

//check if next job  boige is in position [ie. in zone]
	//if so select odd bogie to start then even
	//if not check if other rail is in position
		//if so select
CASE JobCase OF
	0: //Select new GCode File to Execute
	10: //Check RailPriority
		IF RailPriority = 1 AND (SD1State=1 OR SD1State=5) THEN (* in position for SprayA or SprayB *)
			IF SD1State=1 THEN JobCase:=15; END_IF
			IF SD1State=5 THEN JobCase:=25; END_IF
			ELSIF RailPriority =2 AND (SD2State=1 OR SD2State=5) THEN (* in position for SprayA or SprayB *)
				IF SD2State= 1 THEN JobCase:=215; END_IF
				IF SD2State= 5 THEN JobCase:=225; END_IF
			//No movement from this statement until a bogie is in position
		END_IF
	15: //SD1 Prio and in position for SprayA
		IF WX1SprayJob.AKeyDone=0 THEN
			// call WX1SprayJob.AKeyFile 
		END_IF
		IF WX1SPrayJob.AKeyDone AND WX1sprayjob.AMacroDone=0 THEN
			// if AKeyFile Complete then call Macro file
		END_IF
		IF WX1SprayJob.AKeyDone AND WX1SprayJob.AMacroDone THEN
			JobCase:=17; //move to WX2jobs
		END_IF
	17: //SD1 Wx2SprayA
		IF WX2SprayJob.AKeyDone=0 THEN
			// call WX1SprayJob.AKeyFile 
		END_IF
		IF Wx2SPrayJob.AKeyDone AND Wx2sprayjob.AMacroDone=0 THEN
			// if AKeyFile Complete then call Macro file
		END_IF
		IF WX2SprayJob.AKeyDone AND WX2SprayJob.AMacroDone THEN
			JobCase:=0; //move to new selection
		END_IF
		
	25: //SD1 Prio and In position for SprayB
		IF WX1SprayJob.BKeyDone=0 THEN
			// call WX1SprayJob.AKeyFile 
		END_IF
		IF WX1SPrayJob.BKeyDone AND WX1sprayjob.BMacroDone=0 THEN
			// if AKeyFile Complete then call Macro file
		END_IF
		IF WX1SprayJob.BKeyDone AND WX1SprayJob.BMacroDone THEN
			JobCase:=27; //move to WX2jobs
		END_IF
	27: //SD1 WX2 SPrayB
		IF WX2SprayJob.BKeyDone=0 THEN
			// call WX1SprayJob.AKeyFile 
		END_IF
		IF Wx2SPrayJob.BKeyDone AND Wx2sprayjob.BMacroDone=0 THEN
			// if AKeyFile Complete then call Macro file
		END_IF
		IF WX2SprayJob.BKeyDone AND WX2SprayJob.BMacroDone THEN
			JobCase:=0; //move to new selection
		END_IF
	215: //SD2 Prio and in Position for SprayA
	225: //SD2 Prio and in Position for SprayB
END_CASE


CASE nCase OF
	10:
		PLCMachineMode[0].MDI := TRUE;
		nCase := 20;
		
	20:
		IF PRG_CNCChannelHandler.CNCChannel[0].currentmode = 3 THEN
			PLCMachineMode[0].MDIString := Wx4sprayjob.AKeyFile;
			PLCMachineMode[0].Start := TRUE;
			nCase := 30;
		END_IF
	
	30:
		IF PRG_CNCChannelHandler.CNCChannel[0].currentstate = 4 THEN
			nCase := 40;
		END_IF
		
	40:
		IF PRG_CNCChannelHandler.CNCChannel[0].currentstate = 3 THEN
			PLCMachineMode[0].Manual := TRUE;
			nCase := 0;
		END_IF
END_CASE

END_PROGRAM

// ---- Machine System/PRGs/CAM_CNC/myCNC_CureQue.TcPOU
PROGRAM myCNC_CureQue
VAR
END_VAR

END_PROGRAM

// ---- Machine System/PRGs/CAM_CNC/myCNC_JobQue.TcPOU
PROGRAM myCNC_JobQue
VAR

	
END_VAR

END_PROGRAM

// ---- Machine System/PRGs/CAM_CNC/myParts.TcPOU
PROGRAM myParts
VAR
END_VAR

END_PROGRAM

// ---- Machine System/PRGs/DB/PRG_SEQUENCE.TcPOU
PROGRAM PRG_SEQUENCE
VAR
	
	Process			:	ARRAY [1..Max_DBCOLUMNS] OF ST_Process;
	fbSQLDatabase	:	FB_SQLDatabaseEvt (sNetID := '', tTimeout := T#5S);
	fbSQLCommand	:	FB_SQLCommandEvt (sNetID := '', tTimeout := T#5S);
	step			:	INT :=10 ;
	CMD_1			:	STRING(5000);
	CMD_2			:	STRING(5000);
	CMD_3			:	STRING(5000);
	CMD_4			:	STRING(5000);
	sCMD			:	STRING(5000);
	sCMD1			:	STRING(5000);
	sCMD2			:	STRING(5000);
	sCMD3			:	STRING(5000);
	sCMD4			:	STRING(5000);
	sCMD5			:	STRING(5000);
	sCMD6			:	STRING(5000);
	BasketID		:	STRING(5000);
	TotalItem		:	STRING(5000);
	Flavor			:	STRING(5000);
	Id				: int;
	PointId			: STRING(5000);
	XCur			: STRING(5000);
	YCur			: STRING(5000);
	ZCur			: STRING(5000);
	RCur			: STRING(5000);
	VCur			: STRING(5000);
	Dist			: STRING(5000);
	
	

END_VAR

IF GVL_Log.NewMeasure =1 AND GVL_log.ReadytoLog =1 THEN
	GVL_Log.NewMeasure :=0;
	XCur := GVL_Log.XCur;
	YCur := GVL_Log.YCur;
	ZCur := GVL_Log.ZCur;
	RCur := GVL_Log.RCur;
	VCur := GVL_Log.VCur;
	Dist := GVL_Log.Dist;
	step :=10;
	GVL_log.ReadytoLog :=0; //will be reset after getting to step 1031
	Id := Id + 1;
	PointId := INT_TO_STRING(id);
	
	
END_IF
IF GVL_HMI.LogByDis =1 AND GVL_log.ReadytoLog =1 AND GVL_HMI.LogEveryDis >= 1 THEN
	IF ABS(GVL_HMI.LastLogDisX -PRG_CNCAxesHandler.fbCNC_Axis[0].stStatus.fSetPosACS) >= GVL_Hmi.LogEveryDis OR
		ABS(GVL_HMI.LastLogDisY -PRG_CNCAxesHandler.fbCNC_Axis[1].stStatus.fSetPosACS) >= GVL_Hmi.LogEveryDis THEN
	
		XCur := GVL_Log.XCur;
		YCur := GVL_Log.YCur;
		ZCur := GVL_Log.ZCur;
		RCur := GVL_Log.RCur;
		VCur := GVL_Log.VCur;
		Dist := GVL_Log.Dist;
		step :=10;
		GVL_log.ReadytoLog :=0; //will be reset after getting to step 1031
		Id := Id + 1;
		PointId := INT_TO_STRING(id);
		GVL_HMI.LastLogDisX := PRG_CNCAxesHandler.fbCNC_Axis[0].stStatus.fSetPosACS; //last log of X
		GVL_HMI.LastLogDisY := PRG_CNCAxesHandler.fbCNC_Axis[1].stStatus.fSetPosACS; //last log of Y
		END_IF
	
END_IF
CASE step OF
	

	10: //OPEN CONNECTION
		IF fbSQLDatabase.Connect(1) THEN
			step := step + 10;
		END_IF
		
	20: //CREATE COMMAND
		IF fbSQLDatabase.CreateCmd(ADR(fbSQLCommand)) THEN
			step := step + 10;
		END_IF
	
	30: //INSERT COMMAND
		CMD_1 	:= 'INSERT into TwinCATSQL1 (PointID, LoadingTime, XCur, YCur, ZCur, RCur, VCur, Distance) VALUES(';
		CMD_2 	:= ', (CONVERT(varchar(20), GETDATE(),108)), ';
		CMD_3 	:= ')';
		sCMD 	:= CONCAT (CMD_1, CONCAT(PointId, CMD_2));
		sCMD1	:= CONCAT (sCMD, CONCAT(CONCAT('$'',XCur), '$','));
		sCMD2	:= CONCAT (sCMD1, CONCAT(CONCAT('$'',YCur), '$','));
		sCMD3	:= CONCAT (sCMD2, CONCAT(CONCAT('$'',ZCur), '$','));
		sCMD4	:= CONCAT (sCMD3, CONCAT(CONCAT('$'',RCur), '$','));
		sCMD5	:= CONCAT (sCMD4, CONCAT(CONCAT('$'',VCur), '$','));
		sCMD6	:= CONCAT (sCMD5, CONCAT(Dist, CMD_3));
		IF fbSQLCommand.Execute(ADR(sCMD6), SIZEOF(sCMD6)) THEN
			step := step + 1000;
		END_IF
	
	1030: //CLOSE CONNECTION
		IF fbSQLDatabase.Disconnect() THEN
			step := step + 1;
			GVL_Log.PointLogged :=1;
			GVL_Log.ReadytoLog 	:=1;
		END_IF
	
END_CASE

IF GVL_Log.PointLogged =1 THEN
	//message point logged
	ELSE
		//message point log failed try again?
END_IF

END_PROGRAM

// ---- Machine System/PRGs/Mold Laser Mapping/myDistance.TcPOU
PROGRAM myDistance
VAR
	iBaseDist		:	INT;	//baseline distance for calibration 
	iMeasure		:	INT;	//Measured distance
	//prob only need to use the array and not toolmeasure all the time.  Or can push each new toolmeasure into aMeasureArr
	ToolMeasure		: 	Measure;	// Structure of current points during measuring
	aMeasureArr		:	ARRAY [1..2] OF Measure;
	
	myCSV: FB_CSV_RECIPE;
	
	myData :ARRAY [0..1, 0..MAX_CSV_ROWS] OF STRING(MAX_CSV_FIELD_LENGTH);
	
	
END_VAR


//Request z axis goes to home
//Request x and y axis goes to home
//Request a and c axis goes to home

//calibrate sensor to known empty location at home
//if all at home then do this   vvv 


//move to center line of trunnion and Measure off the trunnion base plate
//validate trunnion is centered

//begin measuring tool

//Manual Measure recording process
IF GVL_HMI.MeasureNow = 1 THEN
	GVL_HMI.MeasureNow :=0; //reset for one shot
	ToolMeasure.Dist :=	GVL_io.iDistSens;   
	ToolMeasure.XCur := PRG_CNCAxesHandler.fbCNC_Axis[0].stStatus.fSetPosACS;
	ToolMeasure.YCur := PRG_CNCAxesHandler.fbCNC_Axis[1].stStatus.fSetPosACS;
	ToolMeasure.ZCur := PRG_CNCAxesHandler.fbCNC_Axis[2].stStatus.fSetPosACS;
	ToolMeasure.strX :=LREAL_TO_STRING(ToolMeasure.XCur);
	ToolMeasure.strY :=LREAL_TO_STRING(ToolMeasure.YCur);
	ToolMeasure.strZ :=LREAL_TO_STRING(ToolMeasure.ZCur);
	ToolMeasure.strR :=LREAL_TO_STRING(ToolMeasure.RCur);
	ToolMeasure.strV :=LREAL_TO_STRING(ToolMeasure.VCur);
	GVL_Log.XCur := Toolmeasure.strX;
	GVL_Log.YCur := Toolmeasure.strY;
	GVL_Log.ZCur := Toolmeasure.strZ;
	GVL_Log.RCur := Toolmeasure.strR;
	GVL_Log.VCur := Toolmeasure.strV;
	GVL_log.Dist := INT_TO_STRING(Toolmeasure.Dist);
	GVL_HMI.sMeasurePointDis := Concat(Concat(Concat(ToolMeasure.strX,' , '),Concat(ToolMeasure.strY, ' , ')),(ToolMeasure.strZ));
		GVL_HMI.sMeasurePointDis := concat(GVL_HMI.sMeasurePointDis, ' , ');
		GVL_HMI.sMeasurePointDis := Concat(GVL_HMI.sMeasurePointDis, Concat(ToolMeasure.strR, ' , '));
		GVL_HMI.sMeasurePointDis := Concat(GVL_HMI.sMeasurePointDis, Concat(ToolMeasure.strV, ' , '));
		GVL_HMI.sMeasurePointDis := Concat(GVL_HMI.sMeasurePointDis, GVL_Log.Dist);
	
	GVL_log.NewMeasure :=1;	//log a new measure point it will be turned off in log function
END_IF

IF GVL_HMI.SetReferenceNow = 1 THEN
	GVL_HMI.SetReferenceNow :=0;
	iBaseDist := GVL_io.iDistSens; //Measure off ref surface in this case the round top tube at tallest point
	ToolMeasure.XRef := PRG_CNCAxesHandler.fbCNC_Axis[0].stStatus.fSetPosACS;
	ToolMeasure.YRef := PRG_CNCAxesHandler.fbCNC_Axis[1].stStatus.fSetPosACS;
	ToolMeasure.ZRef := PRG_CNCAxesHandler.fbCNC_Axis[2].stStatus.fSetPosACS;
	ToolMeasure.strX_Ref :=LREAL_TO_STRING(ToolMeasure.XCur);
	ToolMeasure.strY_Ref :=LREAL_TO_STRING(ToolMeasure.YCur);
	ToolMeasure.strZ_Ref :=LREAL_TO_STRING(ToolMeasure.ZCur);
	GVL_HMI.sReferenceDis := Concat(Concat(Concat(ToolMeasure.strX,' , '),Concat(ToolMeasure.strY, ' , ')),(ToolMeasure.strZ));
	GVL_Log.XRef := Toolmeasure.strX;
	GVL_Log.YRef := Toolmeasure.strY;
	GVL_Log.ZRef := Toolmeasure.strZ;
	GVL_Log.RRef := Toolmeasure.strR;
	GVL_Log.VRef := Toolmeasure.strV;
	
	GVL_log.DistRef := INT_TO_STRING(iBaseDist);
	
END_IF

IF GVL_HMI.LogByDis =1 THEN
	ToolMeasure.Dist :=	GVL_io.iDistSens;   
	ToolMeasure.XCur := PRG_CNCAxesHandler.fbCNC_Axis[0].stStatus.fSetPosACS;
	ToolMeasure.YCur := PRG_CNCAxesHandler.fbCNC_Axis[1].stStatus.fSetPosACS;
	ToolMeasure.ZCur := PRG_CNCAxesHandler.fbCNC_Axis[2].stStatus.fSetPosACS;
	ToolMeasure.strX :=LREAL_TO_STRING(ToolMeasure.XCur);
	ToolMeasure.strY :=LREAL_TO_STRING(ToolMeasure.YCur);
	ToolMeasure.strZ :=LREAL_TO_STRING(ToolMeasure.ZCur);
	ToolMeasure.strR :=LREAL_TO_STRING(ToolMeasure.RCur);
	ToolMeasure.strV :=LREAL_TO_STRING(ToolMeasure.VCur);
	GVL_Log.XCur := Toolmeasure.strX;
	GVL_Log.YCur := Toolmeasure.strY;
	GVL_Log.ZCur := Toolmeasure.strZ;
	GVL_Log.RCur := Toolmeasure.strR;
	GVL_Log.VCur := Toolmeasure.strV;
	GVL_log.Dist := INT_TO_STRING(Toolmeasure.Dist);
	GVL_HMI.sMeasurePointDis := Concat(Concat(Concat(ToolMeasure.strX,' , '),Concat(ToolMeasure.strY, ' , ')),(ToolMeasure.strZ));
		GVL_HMI.sMeasurePointDis := concat(GVL_HMI.sMeasurePointDis, ' , ');
		GVL_HMI.sMeasurePointDis := Concat(GVL_HMI.sMeasurePointDis, Concat(ToolMeasure.strR, ' , '));
		GVL_HMI.sMeasurePointDis := Concat(GVL_HMI.sMeasurePointDis, Concat(ToolMeasure.strV, ' , '));
		GVL_HMI.sMeasurePointDis := Concat(GVL_HMI.sMeasurePointDis, GVL_Log.Dist);
	
END_IF
myCSV(
	bReadCSV:= , 
	bWriteCSV:= , 
	sFile:= 'C:\Users\administrator\Desktop\Testcsv.csv', 
	sDelimeter:= , 
	bBusy=> , 
	bErr=> , 
	bReadingDone=> , 
	bWritingDone=>  , 
	arrCSVData:= myData );

END_PROGRAM
